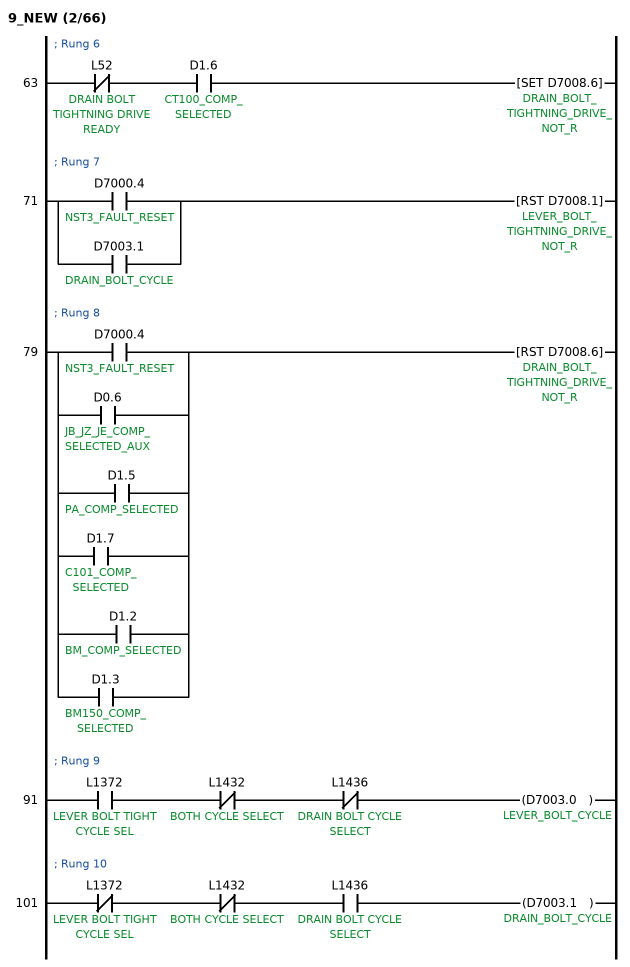
[picture p120: ladder of 9_NEW, rungs at steps 63 to 101]
; Rung 6
63    LDI     L52  ; DRAIN BOLT TIGHTNING DRIVE READY
      AND     D1.6  ; CT100_COMP_SELECTED
      SET     D7008.6  ; DRAIN_BOLT_TIGHTNING_DRIVE_NOT_R
; Rung 7
71    LD      D7000.4  ; NST3_FAULT_RESET
      OR      D7003.1  ; DRAIN_BOLT_CYCLE
      RST     D7008.1  ; LEVER_BOLT_TIGHTNING_DRIVE_NOT_R
; Rung 8
79    LD      D7000.4  ; NST3_FAULT_RESET
      OR      D0.6  ; JB_JZ_JE_COMP_SELECTED_AUX
      OR      D1.5  ; PA_COMP_SELECTED
      OR      D1.7  ; C101_COMP_SELECTED
      OR      D1.2  ; BM_COMP_SELECTED
      OR      D1.3  ; BM150_COMP_SELECTED
      RST     D7008.6  ; DRAIN_BOLT_TIGHTNING_DRIVE_NOT_R
; Rung 9
91    LD      L1372  ; LEVER BOLT TIGHT CYCLE SEL
      ANI     L1432  ; BOTH CYCLE SELECT
      ANI     L1436  ; DRAIN BOLT CYCLE SELECT
      OUT     D7003.0  ; LEVER_BOLT_CYCLE
; Rung 10
101   LDI     L1372  ; LEVER BOLT TIGHT CYCLE SEL
      ANI     L1432  ; BOTH CYCLE SELECT
      AND     L1436  ; DRAIN BOLT CYCLE SELECT
      OUT     D7003.1  ; DRAIN_BOLT_CYCLE
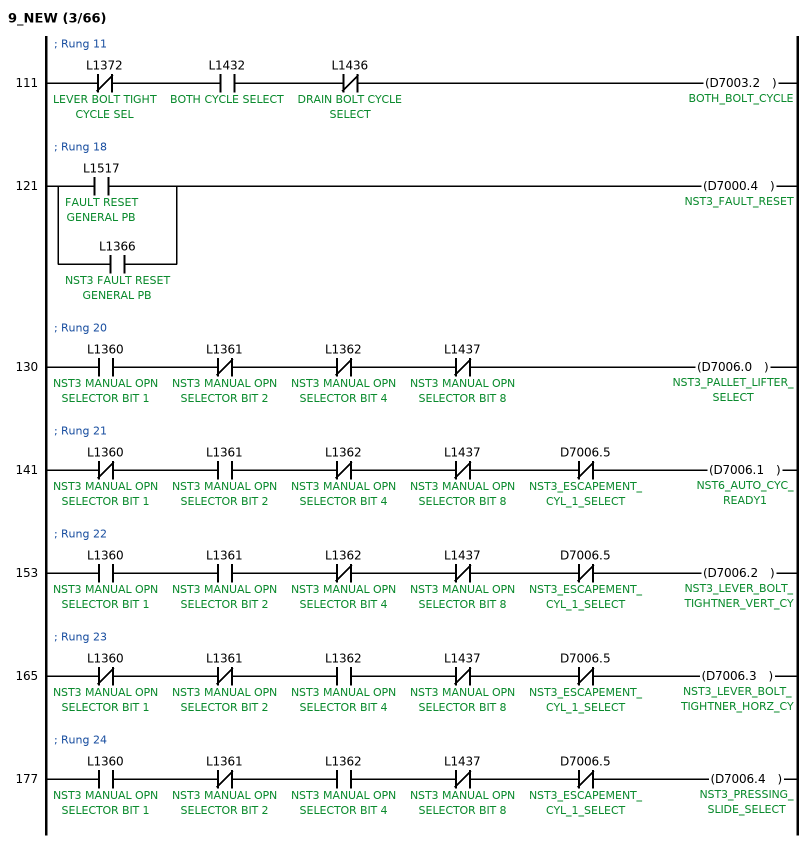
; Rung 11
111   LDI     L1372  ; LEVER BOLT TIGHT CYCLE SEL
      AND     L1432  ; BOTH CYCLE SELECT
      ANI     L1436  ; DRAIN BOLT CYCLE SELECT
      OUT     D7003.2  ; BOTH_BOLT_CYCLE
; Rung 18
121   LD      L1517  ; FAULT RESET GENERAL PB
      OR      L1366  ; NST3 FAULT RESET GENERAL PB
      OUT     D7000.4  ; NST3_FAULT_RESET
; Rung 20
130   LD      L1360  ; NST3 MANUAL OPN SELECTOR BIT 1
      ANI     L1361  ; NST3 MANUAL OPN SELECTOR BIT 2
      ANI     L1362  ; NST3 MANUAL OPN SELECTOR BIT 4
      ANI     L1437  ; NST3 MANUAL OPN SELECTOR BIT 8
      OUT     D7006.0  ; NST3_PALLET_LIFTER_SELECT
; Rung 21
141   LDI     L1360  ; NST3 MANUAL OPN SELECTOR BIT 1
      AND     L1361  ; NST3 MANUAL OPN SELECTOR BIT 2
      ANI     L1362  ; NST3 MANUAL OPN SELECTOR BIT 4
      ANI     L1437  ; NST3 MANUAL OPN SELECTOR BIT 8
      ANI     D7006.5  ; NST3_ESCAPEMENT_CYL_1_SELECT
      OUT     D7006.1  ; NST6_AUTO_CYC_READY1
; Rung 22
153   LD      L1360  ; NST3 MANUAL OPN SELECTOR BIT 1
      AND     L1361  ; NST3 MANUAL OPN SELECTOR BIT 2
      ANI     L1362  ; NST3 MANUAL OPN SELECTOR BIT 4
      ANI     L1437  ; NST3 MANUAL OPN SELECTOR BIT 8
      ANI     D7006.5  ; NST3_ESCAPEMENT_CYL_1_SELECT
      OUT     D7006.2  ; NST3_LEVER_BOLT_TIGHTNER_VERT_CY
; Rung 23
165   LDI     L1360  ; NST3 MANUAL OPN SELECTOR BIT 1
      ANI     L1361  ; NST3 MANUAL OPN SELECTOR BIT 2
      AND     L1362  ; NST3 MANUAL OPN SELECTOR BIT 4
      ANI     L1437  ; NST3 MANUAL OPN SELECTOR BIT 8
      ANI     D7006.5  ; NST3_ESCAPEMENT_CYL_1_SELECT
      OUT     D7006.3  ; NST3_LEVER_BOLT_TIGHTNER_HORZ_CY
; Rung 24
177   LD      L1360  ; NST3 MANUAL OPN SELECTOR BIT 1
      ANI     L1361  ; NST3 MANUAL OPN SELECTOR BIT 2
      AND     L1362  ; NST3 MANUAL OPN SELECTOR BIT 4
      ANI     L1437  ; NST3 MANUAL OPN SELECTOR BIT 8
      ANI     D7006.5  ; NST3_ESCAPEMENT_CYL_1_SELECT
      OUT     D7006.4  ; NST3_PRESSING_SLIDE_SELECT
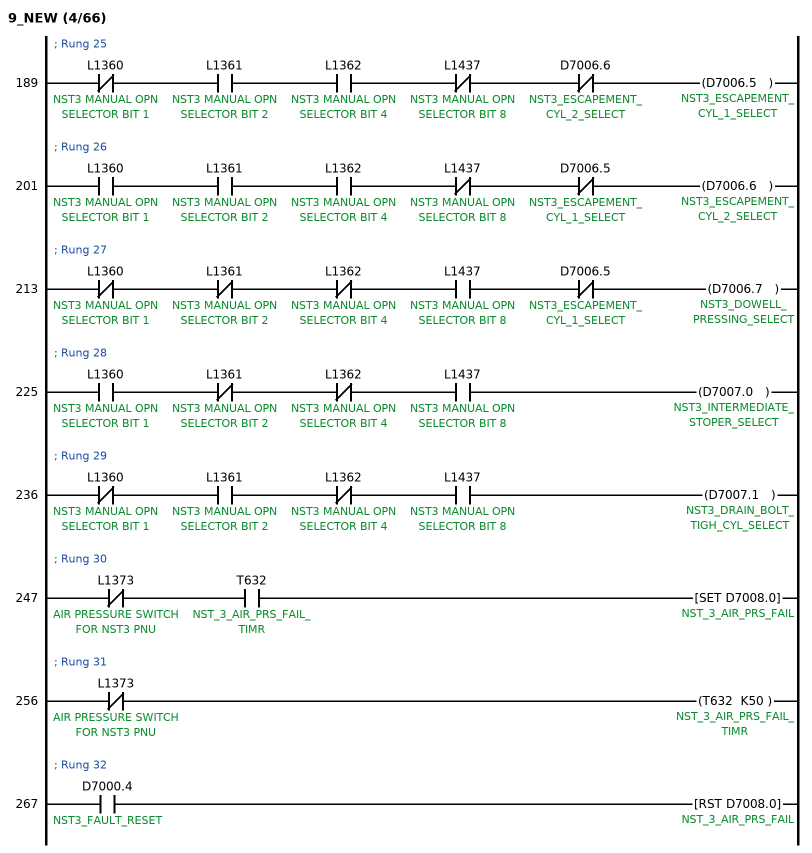
; Rung 25
189   LDI     L1360  ; NST3 MANUAL OPN SELECTOR BIT 1
      AND     L1361  ; NST3 MANUAL OPN SELECTOR BIT 2
      AND     L1362  ; NST3 MANUAL OPN SELECTOR BIT 4
      ANI     L1437  ; NST3 MANUAL OPN SELECTOR BIT 8
      ANI     D7006.6  ; NST3_ESCAPEMENT_CYL_2_SELECT
      OUT     D7006.5  ; NST3_ESCAPEMENT_CYL_1_SELECT
; Rung 26
201   LD      L1360  ; NST3 MANUAL OPN SELECTOR BIT 1
      AND     L1361  ; NST3 MANUAL OPN SELECTOR BIT 2
      AND     L1362  ; NST3 MANUAL OPN SELECTOR BIT 4
      ANI     L1437  ; NST3 MANUAL OPN SELECTOR BIT 8
      ANI     D7006.5  ; NST3_ESCAPEMENT_CYL_1_SELECT
      OUT     D7006.6  ; NST3_ESCAPEMENT_CYL_2_SELECT
; Rung 27
213   LDI     L1360  ; NST3 MANUAL OPN SELECTOR BIT 1
      ANI     L1361  ; NST3 MANUAL OPN SELECTOR BIT 2
      ANI     L1362  ; NST3 MANUAL OPN SELECTOR BIT 4
      AND     L1437  ; NST3 MANUAL OPN SELECTOR BIT 8
      ANI     D7006.5  ; NST3_ESCAPEMENT_CYL_1_SELECT
      OUT     D7006.7  ; NST3_DOWELL_PRESSING_SELECT
; Rung 28
225   LD      L1360  ; NST3 MANUAL OPN SELECTOR BIT 1
      ANI     L1361  ; NST3 MANUAL OPN SELECTOR BIT 2
      ANI     L1362  ; NST3 MANUAL OPN SELECTOR BIT 4
      AND     L1437  ; NST3 MANUAL OPN SELECTOR BIT 8
      OUT     D7007.0  ; NST3_INTERMEDIATE_STOPER_SELECT
; Rung 29
236   LDI     L1360  ; NST3 MANUAL OPN SELECTOR BIT 1
      AND     L1361  ; NST3 MANUAL OPN SELECTOR BIT 2
      ANI     L1362  ; NST3 MANUAL OPN SELECTOR BIT 4
      AND     L1437  ; NST3 MANUAL OPN SELECTOR BIT 8
      OUT     D7007.1  ; NST3_DRAIN_BOLT_TIGH_CYL_SELECT
; Rung 30
247   LDI     L1373  ; AIR PRESSURE SWITCH FOR NST3 PNU
      AND     T632  ; NST_3_AIR_PRS_FAIL_TIMR
      SET     D7008.0  ; NST_3_AIR_PRS_FAIL
; Rung 31
256   LDI     L1373  ; AIR PRESSURE SWITCH FOR NST3 PNU
      OUT     T632 K50  ; NST_3_AIR_PRS_FAIL_TIMR
; Rung 32
267   LD      D7000.4  ; NST3_FAULT_RESET
      RST     D7008.0  ; NST_3_AIR_PRS_FAIL
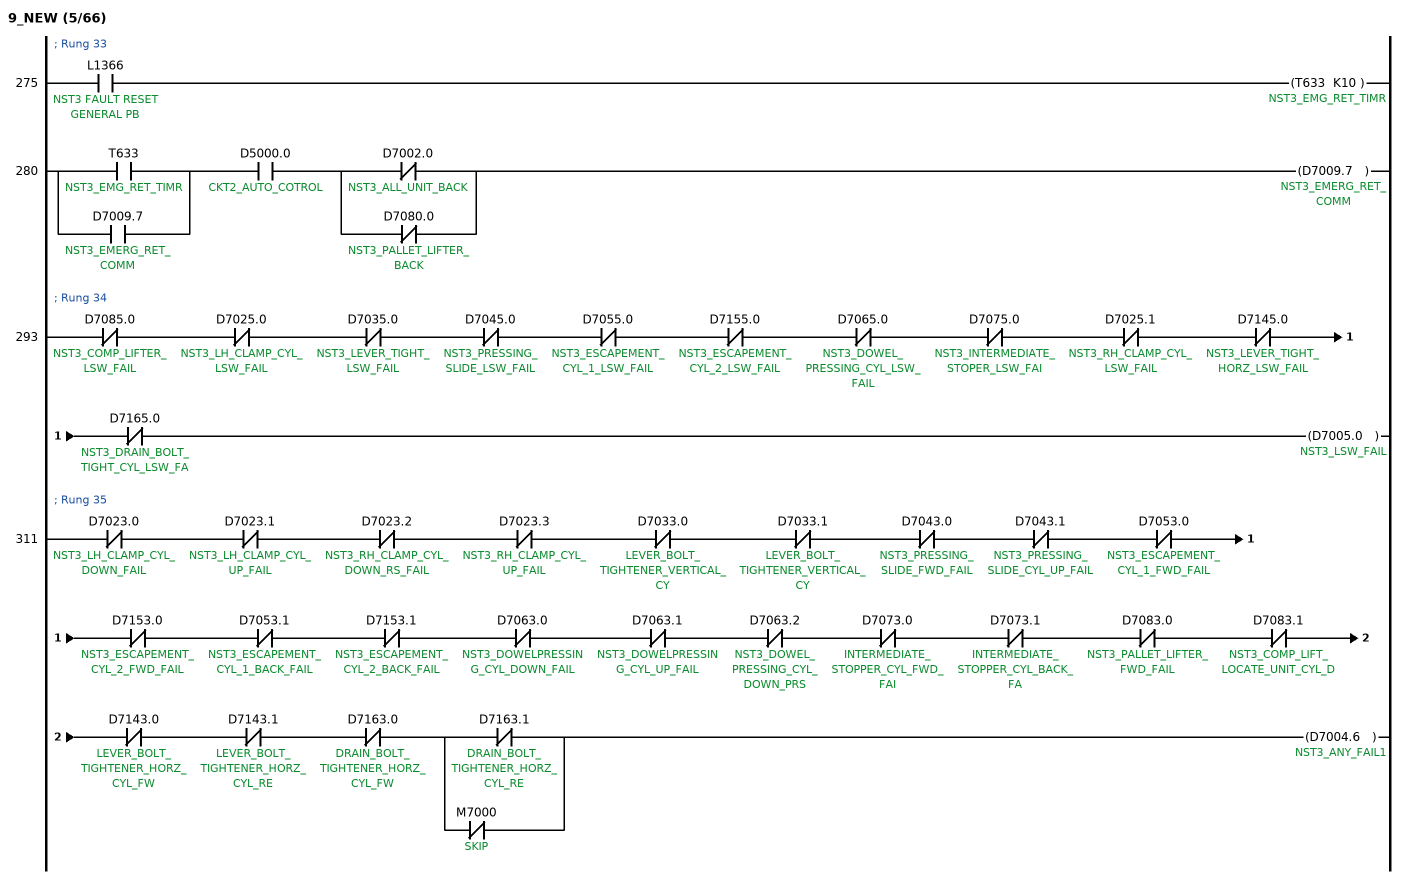
; Rung 33
275   LD      L1366  ; NST3 FAULT RESET GENERAL PB
      OUT     T633 K10  ; NST3_EMG_RET_TIMR
280   LD      T633  ; NST3_EMG_RET_TIMR
      OR      D7009.7  ; NST3_EMERG_RET_COMM
      AND     D5000.0  ; CKT2_AUTO_COTROL
      LDI     D7002.0  ; NST3_ALL_UNIT_BACK
      ORI     D7080.0  ; NST3_PALLET_LIFTER_BACK
      ANB
      OUT     D7009.7  ; NST3_EMERG_RET_COMM
; Rung 34
293   LDI     D7085.0  ; NST3_COMP_LIFTER_LSW_FAIL
      ANI     D7025.0  ; NST3_LH_CLAMP_CYL_LSW_FAIL
      ANI     D7035.0  ; NST3_LEVER_TIGHT_LSW_FAIL
      ANI     D7045.0  ; NST3_PRESSING_SLIDE_LSW_FAIL
      ANI     D7055.0  ; NST3_ESCAPEMENT_CYL_1_LSW_FAIL
      ANI     D7155.0  ; NST3_ESCAPEMENT_CYL_2_LSW_FAIL
      ANI     D7065.0  ; NST3_DOWEL_PRESSING_CYL_LSW_FAIL
      ANI     D7075.0  ; NST3_INTERMEDIATE_STOPER_LSW_FAI
      ANI     D7025.1  ; NST3_RH_CLAMP_CYL_LSW_FAIL
      ANI     D7145.0  ; NST3_LEVER_TIGHT_HORZ_LSW_FAIL
      ANI     D7165.0  ; NST3_DRAIN_BOLT_TIGHT_CYL_LSW_FA
      OUT     D7005.0  ; NST3_LSW_FAIL
; Rung 35
311   LDI     D7023.0  ; NST3_LH_CLAMP_CYL_DOWN_FAIL
      ANI     D7023.1  ; NST3_LH_CLAMP_CYL_UP_FAIL
      ANI     D7023.2  ; NST3_RH_CLAMP_CYL_DOWN_RS_FAIL
      ANI     D7023.3  ; NST3_RH_CLAMP_CYL_UP_FAIL
      ANI     D7033.0  ; LEVER_BOLT_TIGHTENER_VERTICAL_CY
      ANI     D7033.1  ; LEVER_BOLT_TIGHTENER_VERTICAL_CY
      ANI     D7043.0  ; NST3_PRESSING_SLIDE_FWD_FAIL
      ANI     D7043.1  ; NST3_PRESSING_SLIDE_CYL_UP_FAIL
      ANI     D7053.0  ; NST3_ESCAPEMENT_CYL_1_FWD_FAIL
      ANI     D7153.0  ; NST3_ESCAPEMENT_CYL_2_FWD_FAIL
      ANI     D7053.1  ; NST3_ESCAPEMENT_CYL_1_BACK_FAIL
      ANI     D7153.1  ; NST3_ESCAPEMENT_CYL_2_BACK_FAIL
      ANI     D7063.0  ; NST3_DOWELPRESSING_CYL_DOWN_FAIL
      ANI     D7063.1  ; NST3_DOWELPRESSING_CYL_UP_FAIL
      ANI     D7063.2  ; NST3_DOWEL_PRESSING_CYL_DOWN_PRS
      ANI     D7073.0  ; INTERMEDIATE_STOPPER_CYL_FWD_FAI
      ANI     D7073.1  ; INTERMEDIATE_STOPPER_CYL_BACK_FA
      ANI     D7083.0  ; NST3_PALLET_LIFTER_FWD_FAIL
      ANI     D7083.1  ; NST3_COMP_LIFT_LOCATE_UNIT_CYL_D
      ANI     D7143.0  ; LEVER_BOLT_TIGHTENER_HORZ_CYL_FW
      ANI     D7143.1  ; LEVER_BOLT_TIGHTENER_HORZ_CYL_RE
      ANI     D7163.0  ; DRAIN_BOLT_TIGHTENER_HORZ_CYL_FW
      LDI     D7163.1  ; DRAIN_BOLT_TIGHTENER_HORZ_CYL_RE
      ORI     M7000  ; SKIP
      ANB
      OUT     D7004.6  ; NST3_ANY_FAIL1
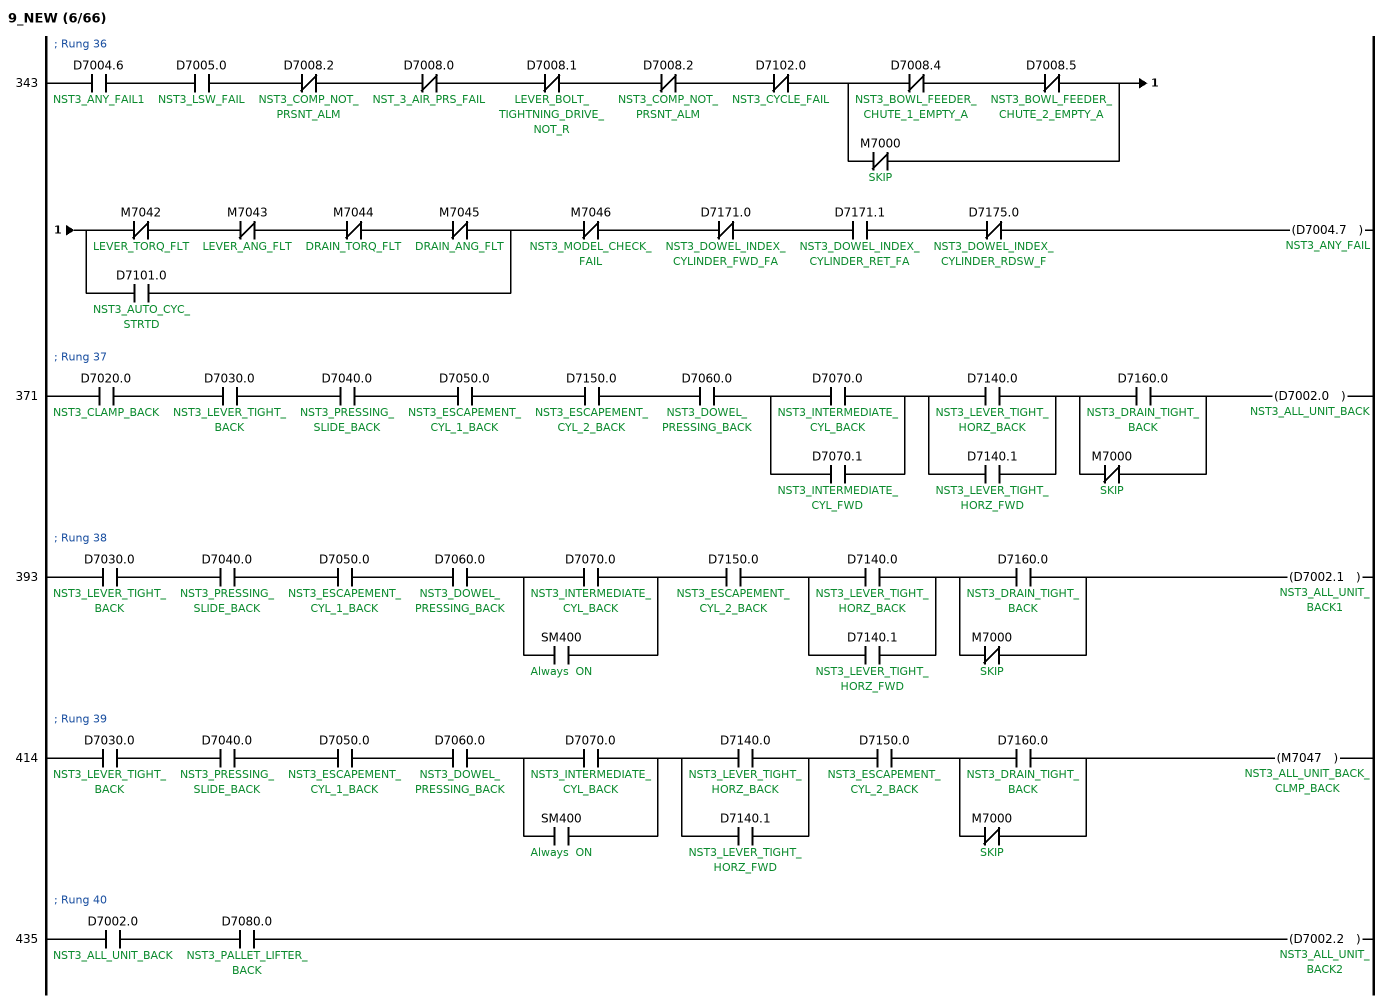
; Rung 36
343   LD      D7004.6  ; NST3_ANY_FAIL1
      AND     D7005.0  ; NST3_LSW_FAIL
      ANI     D7008.2  ; NST3_COMP_NOT_PRSNT_ALM
      ANI     D7008.0  ; NST_3_AIR_PRS_FAIL
      ANI     D7008.1  ; LEVER_BOLT_TIGHTNING_DRIVE_NOT_R
      ANI     D7008.2  ; NST3_COMP_NOT_PRSNT_ALM
      ANI     D7102.0  ; NST3_CYCLE_FAIL
      LDI     D7008.4  ; NST3_BOWL_FEEDER_CHUTE_1_EMPTY_A
      ANI     D7008.5  ; NST3_BOWL_FEEDER_CHUTE_2_EMPTY_A
      ORI     M7000  ; SKIP
      ANB
      LDI     M7042  ; LEVER_TORQ_FLT
      ANI     M7043  ; LEVER_ANG_FLT
      ANI     M7044  ; DRAIN_TORQ_FLT
      ANI     M7045  ; DRAIN_ANG_FLT
      OR      D7101.0  ; NST3_AUTO_CYC_STRTD
      ANB
      ANI     M7046  ; NST3_MODEL_CHECK_FAIL
      ANI     D7171.0  ; NST3_DOWEL_INDEX_CYLINDER_FWD_FA
      AND     D7171.1  ; NST3_DOWEL_INDEX_CYLINDER_RET_FA
      ANI     D7175.0  ; NST3_DOWEL_INDEX_CYLINDER_RDSW_F
      OUT     D7004.7  ; NST3_ANY_FAIL
; Rung 37
371   LD      D7020.0  ; NST3_CLAMP_BACK
      AND     D7030.0  ; NST3_LEVER_TIGHT_BACK
      AND     D7040.0  ; NST3_PRESSING_SLIDE_BACK
      AND     D7050.0  ; NST3_ESCAPEMENT_CYL_1_BACK
      AND     D7150.0  ; NST3_ESCAPEMENT_CYL_2_BACK
      AND     D7060.0  ; NST3_DOWEL_PRESSING_BACK
      LD      D7070.0  ; NST3_INTERMEDIATE_CYL_BACK
      OR      D7070.1  ; NST3_INTERMEDIATE_CYL_FWD
      ANB
      LD      D7140.0  ; NST3_LEVER_TIGHT_HORZ_BACK
      OR      D7140.1  ; NST3_LEVER_TIGHT_HORZ_FWD
      ANB
      LD      D7160.0  ; NST3_DRAIN_TIGHT_BACK
      ORI     M7000  ; SKIP
      ANB
      OUT     D7002.0  ; NST3_ALL_UNIT_BACK
; Rung 38
393   LD      D7030.0  ; NST3_LEVER_TIGHT_BACK
      AND     D7040.0  ; NST3_PRESSING_SLIDE_BACK
      AND     D7050.0  ; NST3_ESCAPEMENT_CYL_1_BACK
      AND     D7060.0  ; NST3_DOWEL_PRESSING_BACK
      LD      D7070.0  ; NST3_INTERMEDIATE_CYL_BACK
      OR      SM400  ; Always  ON
      ANB
      AND     D7150.0  ; NST3_ESCAPEMENT_CYL_2_BACK
      LD      D7140.0  ; NST3_LEVER_TIGHT_HORZ_BACK
      OR      D7140.1  ; NST3_LEVER_TIGHT_HORZ_FWD
      ANB
      LD      D7160.0  ; NST3_DRAIN_TIGHT_BACK
      ORI     M7000  ; SKIP
      ANB
      OUT     D7002.1  ; NST3_ALL_UNIT_BACK1
; Rung 39
414   LD      D7030.0  ; NST3_LEVER_TIGHT_BACK
      AND     D7040.0  ; NST3_PRESSING_SLIDE_BACK
      AND     D7050.0  ; NST3_ESCAPEMENT_CYL_1_BACK
      AND     D7060.0  ; NST3_DOWEL_PRESSING_BACK
      LD      D7070.0  ; NST3_INTERMEDIATE_CYL_BACK
      OR      SM400  ; Always  ON
      ANB
      LD      D7140.0  ; NST3_LEVER_TIGHT_HORZ_BACK
      OR      D7140.1  ; NST3_LEVER_TIGHT_HORZ_FWD
      ANB
      AND     D7150.0  ; NST3_ESCAPEMENT_CYL_2_BACK
      LD      D7160.0  ; NST3_DRAIN_TIGHT_BACK
      ORI     M7000  ; SKIP
      ANB
      OUT     M7047  ; NST3_ALL_UNIT_BACK_CLMP_BACK
; Rung 40
435   LD      D7002.0  ; NST3_ALL_UNIT_BACK
      AND     D7080.0  ; NST3_PALLET_LIFTER_BACK
      OUT     D7002.2  ; NST3_ALL_UNIT_BACK2
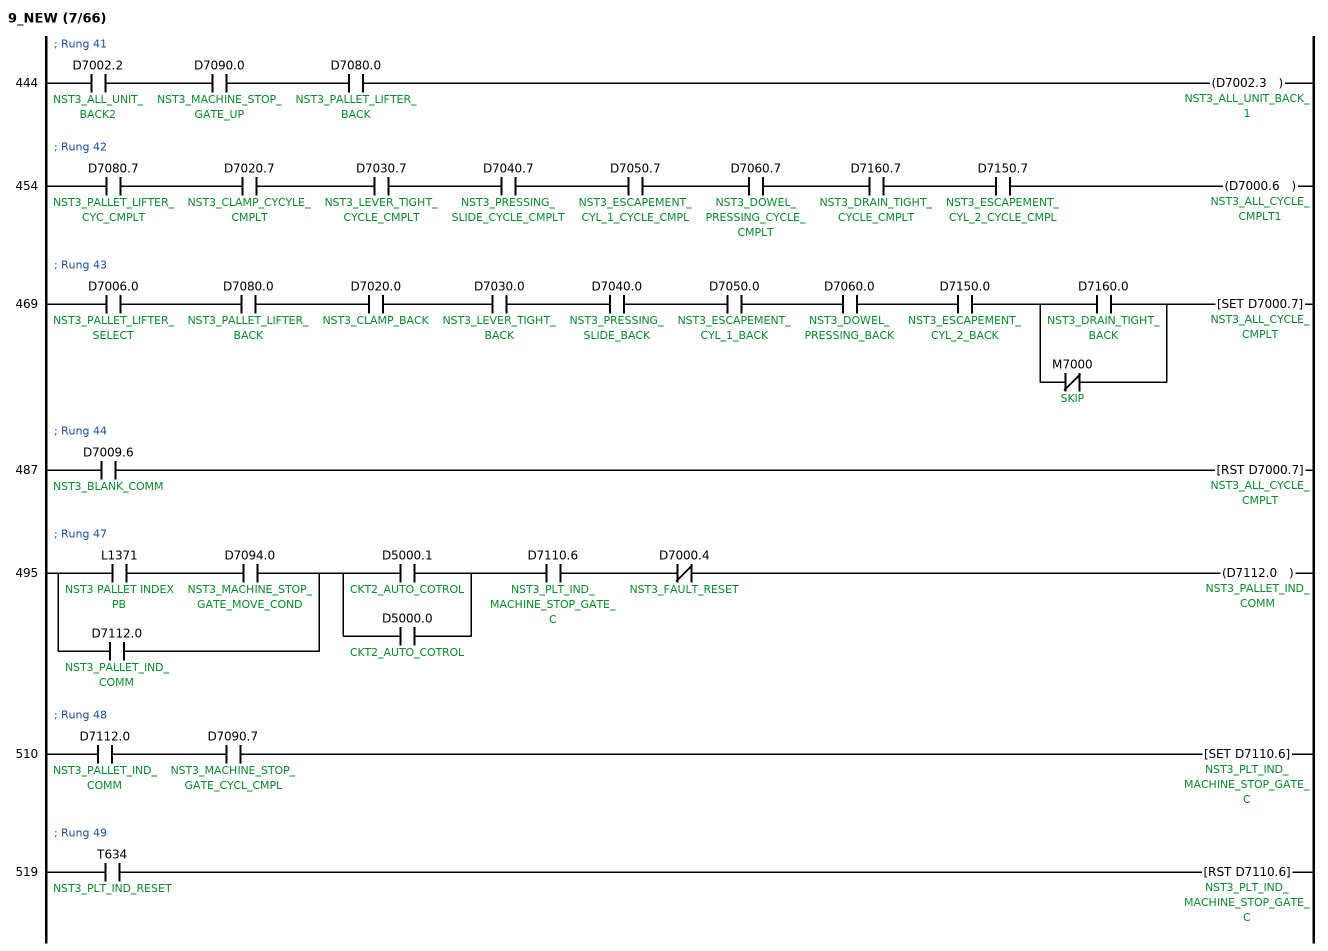
; Rung 41
444   LD      D7002.2  ; NST3_ALL_UNIT_BACK2
      AND     D7090.0  ; NST3_MACHINE_STOP_GATE_UP
      AND     D7080.0  ; NST3_PALLET_LIFTER_BACK
      OUT     D7002.3  ; NST3_ALL_UNIT_BACK_1
; Rung 42
454   LD      D7080.7  ; NST3_PALLET_LIFTER_CYC_CMPLT
      AND     D7020.7  ; NST3_CLAMP_CYCYLE_CMPLT
      AND     D7030.7  ; NST3_LEVER_TIGHT_CYCLE_CMPLT
      AND     D7040.7  ; NST3_PRESSING_SLIDE_CYCLE_CMPLT
      AND     D7050.7  ; NST3_ESCAPEMENT_CYL_1_CYCLE_CMPL
      AND     D7060.7  ; NST3_DOWEL_PRESSING_CYCLE_CMPLT
      AND     D7160.7  ; NST3_DRAIN_TIGHT_CYCLE_CMPLT
      AND     D7150.7  ; NST3_ESCAPEMENT_CYL_2_CYCLE_CMPL
      OUT     D7000.6  ; NST3_ALL_CYCLE_CMPLT1
; Rung 43
469   LD      D7006.0  ; NST3_PALLET_LIFTER_SELECT
      AND     D7080.0  ; NST3_PALLET_LIFTER_BACK
      AND     D7020.0  ; NST3_CLAMP_BACK
      AND     D7030.0  ; NST3_LEVER_TIGHT_BACK
      AND     D7040.0  ; NST3_PRESSING_SLIDE_BACK
      AND     D7050.0  ; NST3_ESCAPEMENT_CYL_1_BACK
      AND     D7060.0  ; NST3_DOWEL_PRESSING_BACK
      AND     D7150.0  ; NST3_ESCAPEMENT_CYL_2_BACK
      LD      D7160.0  ; NST3_DRAIN_TIGHT_BACK
      ORI     M7000  ; SKIP
      ANB
      SET     D7000.7  ; NST3_ALL_CYCLE_CMPLT
; Rung 44
487   LD      D7009.6  ; NST3_BLANK_COMM
      RST     D7000.7  ; NST3_ALL_CYCLE_CMPLT
; Rung 47
495   LD      L1371  ; NST3 PALLET INDEX PB
      AND     D7094.0  ; NST3_MACHINE_STOP_GATE_MOVE_COND
      OR      D7112.0  ; NST3_PALLET_IND_COMM
      LD      D5000.1  ; CKT2_AUTO_COTROL
      OR      D5000.0  ; CKT2_AUTO_COTROL
      ANB
      AND     D7110.6  ; NST3_PLT_IND_MACHINE_STOP_GATE_C
      ANI     D7000.4  ; NST3_FAULT_RESET
      OUT     D7112.0  ; NST3_PALLET_IND_COMM
; Rung 48
510   LD      D7112.0  ; NST3_PALLET_IND_COMM
      AND     D7090.7  ; NST3_MACHINE_STOP_GATE_CYCL_CMPL
      SET     D7110.6  ; NST3_PLT_IND_MACHINE_STOP_GATE_C
; Rung 49
519   LD      T634  ; NST3_PLT_IND_RESET
      RST     D7110.6  ; NST3_PLT_IND_MACHINE_STOP_GATE_C
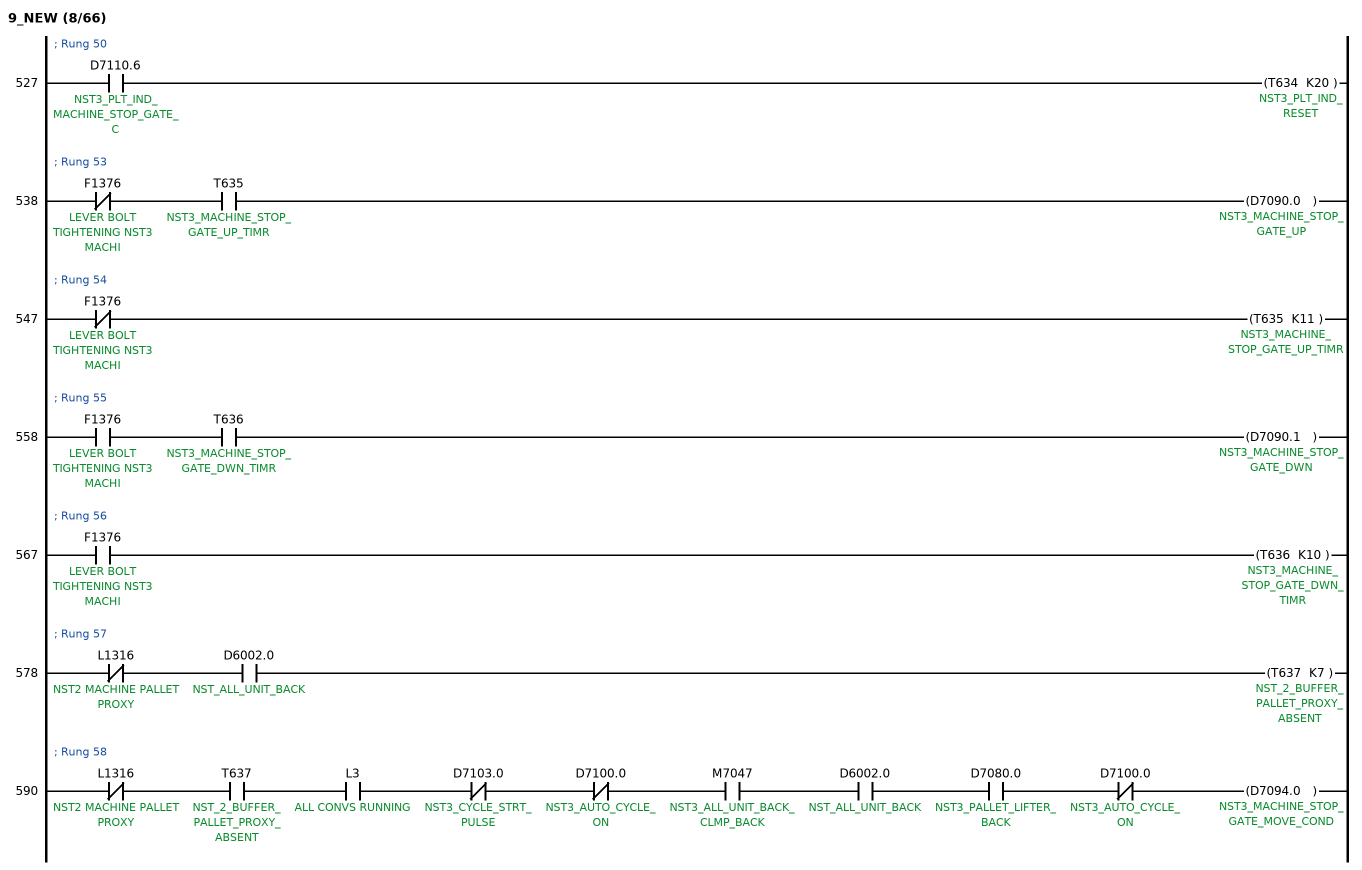
; Rung 50
527   LD      D7110.6  ; NST3_PLT_IND_MACHINE_STOP_GATE_C
      OUT     T634 K20  ; NST3_PLT_IND_RESET
; Rung 53
538   LDI     F1376  ; LEVER BOLT TIGHTENING NST3 MACHI
      AND     T635  ; NST3_MACHINE_STOP_GATE_UP_TIMR
      OUT     D7090.0  ; NST3_MACHINE_STOP_GATE_UP
; Rung 54
547   LDI     F1376  ; LEVER BOLT TIGHTENING NST3 MACHI
      OUT     T635 K11  ; NST3_MACHINE_STOP_GATE_UP_TIMR
; Rung 55
558   LD      F1376  ; LEVER BOLT TIGHTENING NST3 MACHI
      AND     T636  ; NST3_MACHINE_STOP_GATE_DWN_TIMR
      OUT     D7090.1  ; NST3_MACHINE_STOP_GATE_DWN
; Rung 56
567   LD      F1376  ; LEVER BOLT TIGHTENING NST3 MACHI
      OUT     T636 K10  ; NST3_MACHINE_STOP_GATE_DWN_TIMR
; Rung 57
578   LDI     L1316  ; NST2 MACHINE PALLET PROXY
      AND     D6002.0  ; NST_ALL_UNIT_BACK
      OUT     T637 K7  ; NST_2_BUFFER_PALLET_PROXY_ABSENT
; Rung 58
590   LDI     L1316  ; NST2 MACHINE PALLET PROXY
      AND     T637  ; NST_2_BUFFER_PALLET_PROXY_ABSENT
      AND     L3  ; ALL CONVS RUNNING
      ANI     D7103.0  ; NST3_CYCLE_STRT_PULSE
      ANI     D7100.0  ; NST3_AUTO_CYCLE_ON
      AND     M7047  ; NST3_ALL_UNIT_BACK_CLMP_BACK
      AND     D6002.0  ; NST_ALL_UNIT_BACK
      AND     D7080.0  ; NST3_PALLET_LIFTER_BACK
      ANI     D7100.0  ; NST3_AUTO_CYCLE_ON
      OUT     D7094.0  ; NST3_MACHINE_STOP_GATE_MOVE_COND
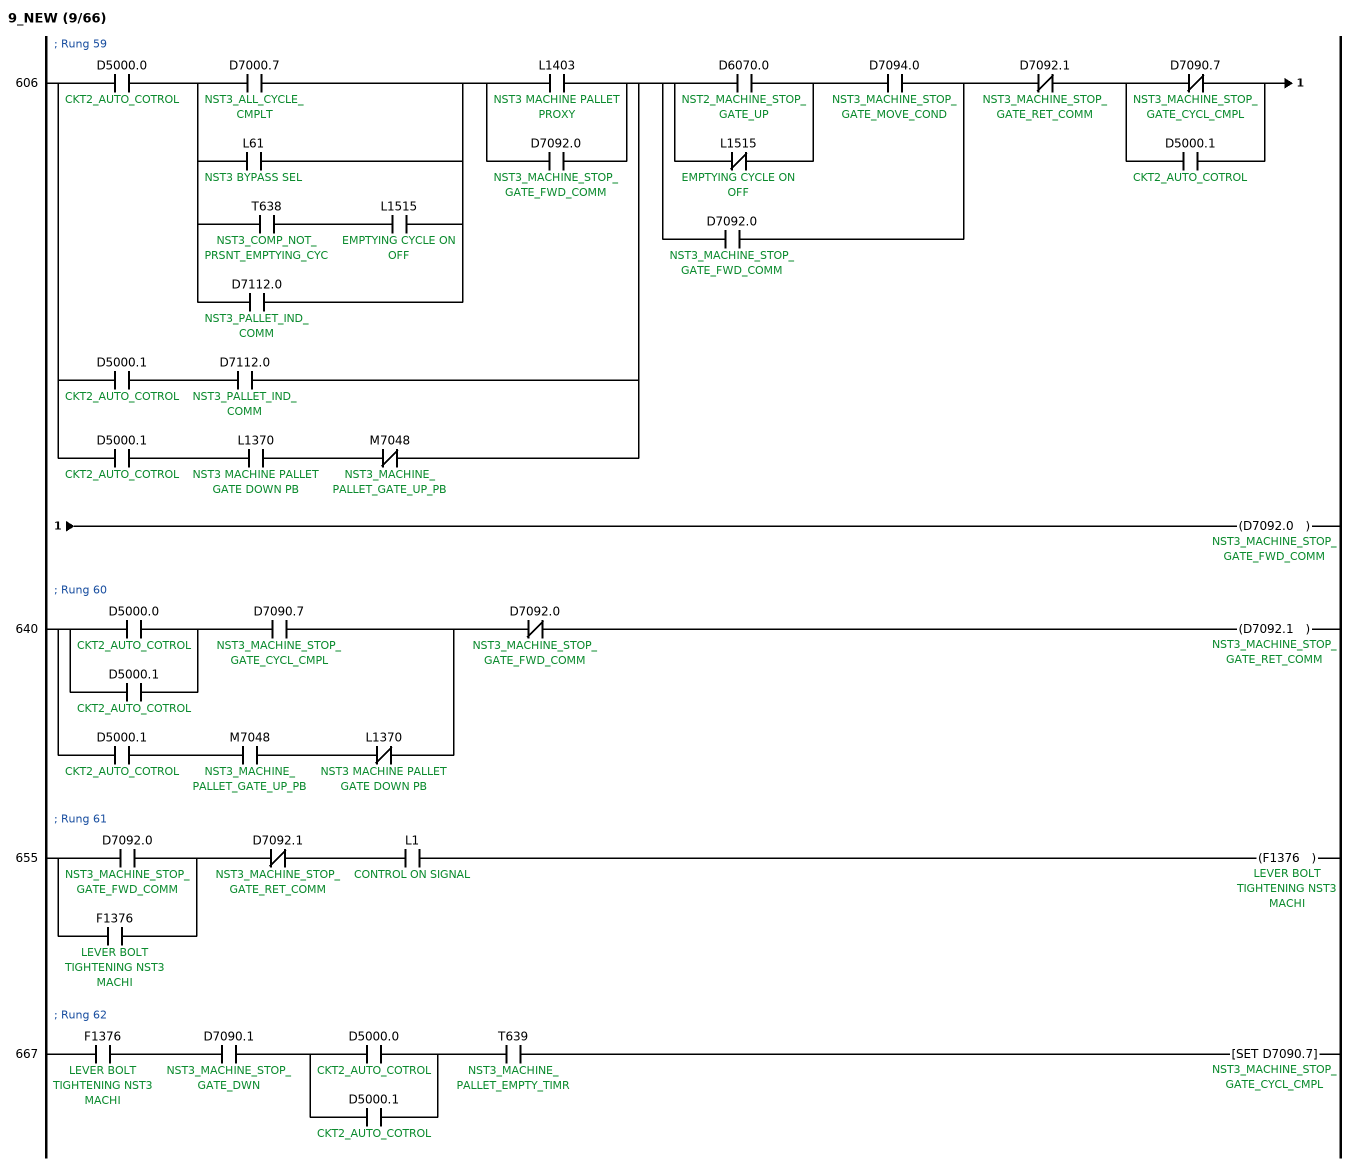
; Rung 59
606   LD      D5000.0  ; CKT2_AUTO_COTROL
      LD      D7000.7  ; NST3_ALL_CYCLE_CMPLT
      OR      L61  ; NST3 BYPASS SEL
      LD      T638  ; NST3_COMP_NOT_PRSNT_EMPTYING_CYC
      AND     L1515  ; EMPTYING CYCLE ON OFF
      ORB
      OR      D7112.0  ; NST3_PALLET_IND_COMM
      ANB
      LD      L1403  ; NST3 MACHINE PALLET PROXY
      OR      D7092.0  ; NST3_MACHINE_STOP_GATE_FWD_COMM
      ANB
      LD      D5000.1  ; CKT2_AUTO_COTROL
      AND     D7112.0  ; NST3_PALLET_IND_COMM
      ORB
      LD      D5000.1  ; CKT2_AUTO_COTROL
      AND     L1370  ; NST3 MACHINE PALLET GATE DOWN PB
      ANI     M7048  ; NST3_MACHINE_PALLET_GATE_UP_PB
      ORB
      LD      D6070.0  ; NST2_MACHINE_STOP_GATE_UP
      ORI     L1515  ; EMPTYING CYCLE ON OFF
      AND     D7094.0  ; NST3_MACHINE_STOP_GATE_MOVE_COND
      OR      D7092.0  ; NST3_MACHINE_STOP_GATE_FWD_COMM
      ANB
      ANI     D7092.1  ; NST3_MACHINE_STOP_GATE_RET_COMM
      LDI     D7090.7  ; NST3_MACHINE_STOP_GATE_CYCL_CMPL
      OR      D5000.1  ; CKT2_AUTO_COTROL
      ANB
      OUT     D7092.0  ; NST3_MACHINE_STOP_GATE_FWD_COMM
; Rung 60
640   LD      D5000.0  ; CKT2_AUTO_COTROL
      OR      D5000.1  ; CKT2_AUTO_COTROL
      AND     D7090.7  ; NST3_MACHINE_STOP_GATE_CYCL_CMPL
      LD      D5000.1  ; CKT2_AUTO_COTROL
      AND     M7048  ; NST3_MACHINE_PALLET_GATE_UP_PB
      ANI     L1370  ; NST3 MACHINE PALLET GATE DOWN PB
      ORB
      ANI     D7092.0  ; NST3_MACHINE_STOP_GATE_FWD_COMM
      OUT     D7092.1  ; NST3_MACHINE_STOP_GATE_RET_COMM
; Rung 61
655   LD      D7092.0  ; NST3_MACHINE_STOP_GATE_FWD_COMM
      OR      F1376  ; LEVER BOLT TIGHTENING NST3 MACHI
      ANI     D7092.1  ; NST3_MACHINE_STOP_GATE_RET_COMM
      AND     L1  ; CONTROL ON SIGNAL
      OUT     F1376  ; LEVER BOLT TIGHTENING NST3 MACHI
; Rung 62
667   LD      F1376  ; LEVER BOLT TIGHTENING NST3 MACHI
      AND     D7090.1  ; NST3_MACHINE_STOP_GATE_DWN
      LD      D5000.0  ; CKT2_AUTO_COTROL
      OR      D5000.1  ; CKT2_AUTO_COTROL
      ANB
      AND     T639  ; NST3_MACHINE_PALLET_EMPTY_TIMR
      SET     D7090.7  ; NST3_MACHINE_STOP_GATE_CYCL_CMPL
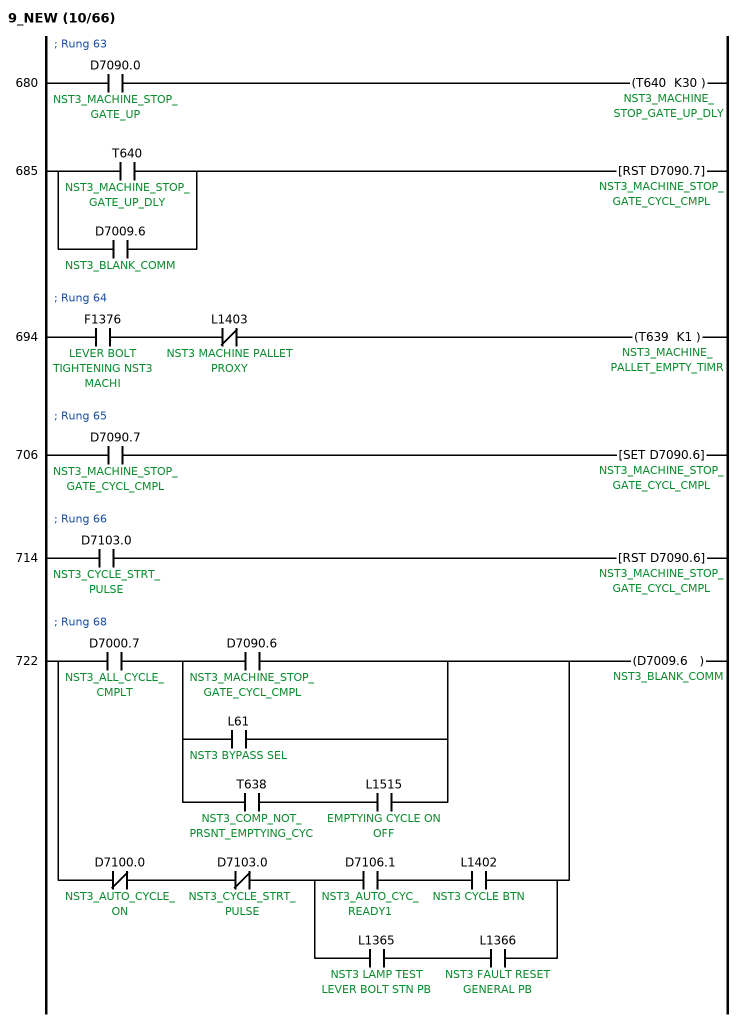
; Rung 63
680   LD      D7090.0  ; NST3_MACHINE_STOP_GATE_UP
      OUT     T640 K30  ; NST3_MACHINE_STOP_GATE_UP_DLY
685   LD      T640  ; NST3_MACHINE_STOP_GATE_UP_DLY
      OR      D7009.6  ; NST3_BLANK_COMM
      RST     D7090.7  ; NST3_MACHINE_STOP_GATE_CYCL_CMPL
; Rung 64
694   LD      F1376  ; LEVER BOLT TIGHTENING NST3 MACHI
      ANI     L1403  ; NST3 MACHINE PALLET PROXY
      OUT     T639 K1  ; NST3_MACHINE_PALLET_EMPTY_TIMR
; Rung 65
706   LD      D7090.7  ; NST3_MACHINE_STOP_GATE_CYCL_CMPL
      SET     D7090.6  ; NST3_MACHINE_STOP_GATE_CYCL_CMPL
; Rung 66
714   LD      D7103.0  ; NST3_CYCLE_STRT_PULSE
      RST     D7090.6  ; NST3_MACHINE_STOP_GATE_CYCL_CMPL
; Rung 68
722   LD      D7000.7  ; NST3_ALL_CYCLE_CMPLT
      LD      D7090.6  ; NST3_MACHINE_STOP_GATE_CYCL_CMPL
      OR      L61  ; NST3 BYPASS SEL
      LD      T638  ; NST3_COMP_NOT_PRSNT_EMPTYING_CYC
      AND     L1515  ; EMPTYING CYCLE ON OFF
      ORB
      ANB
      LDI     D7100.0  ; NST3_AUTO_CYCLE_ON
      ANI     D7103.0  ; NST3_CYCLE_STRT_PULSE
      LD      D7106.1  ; NST3_AUTO_CYC_READY1
      AND     L1402  ; NST3 CYCLE BTN
      LD      L1365  ; NST3 LAMP TEST LEVER BOLT STN PB
      AND     L1366  ; NST3 FAULT RESET GENERAL PB
      ORB
      ANB
      ORB
      OUT     D7009.6  ; NST3_BLANK_COMM
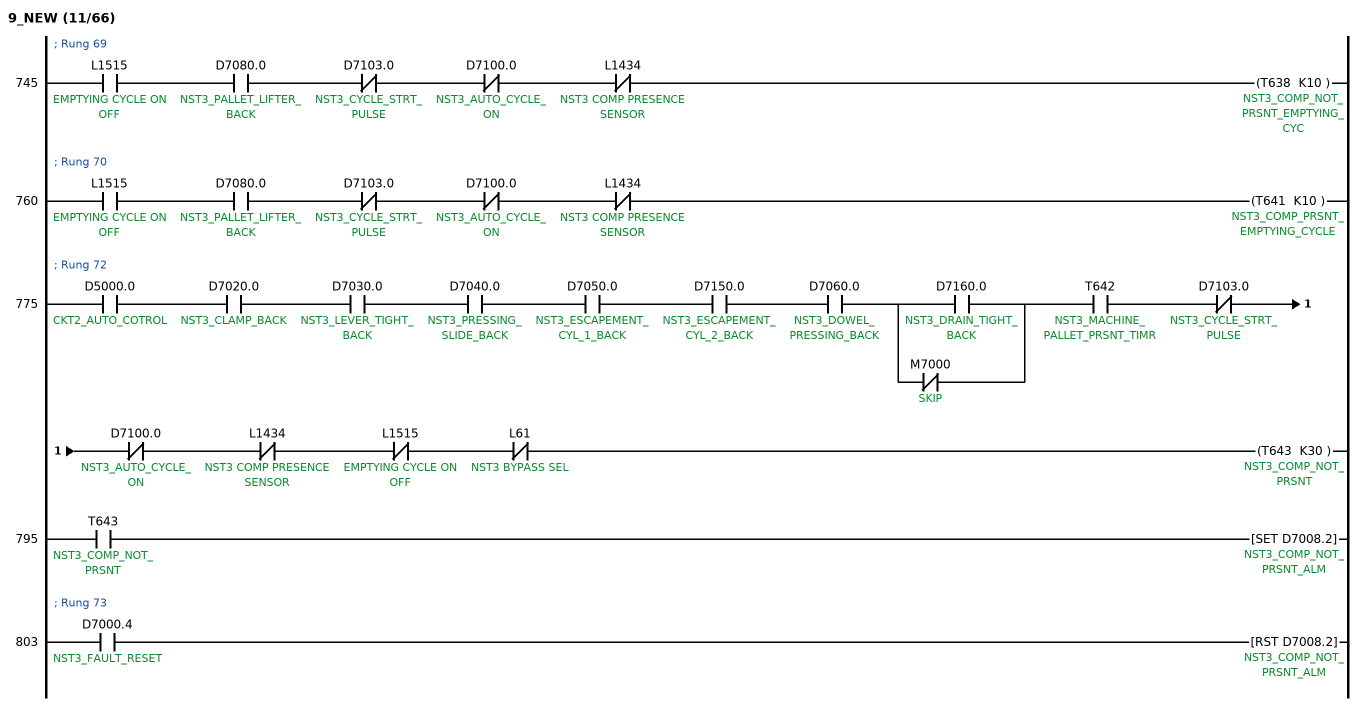
; Rung 69
745   LD      L1515  ; EMPTYING CYCLE ON OFF
      AND     D7080.0  ; NST3_PALLET_LIFTER_BACK
      ANI     D7103.0  ; NST3_CYCLE_STRT_PULSE
      ANI     D7100.0  ; NST3_AUTO_CYCLE_ON
      ANI     L1434  ; NST3 COMP PRESENCE SENSOR
      OUT     T638 K10  ; NST3_COMP_NOT_PRSNT_EMPTYING_CYC
; Rung 70
760   LD      L1515  ; EMPTYING CYCLE ON OFF
      AND     D7080.0  ; NST3_PALLET_LIFTER_BACK
      ANI     D7103.0  ; NST3_CYCLE_STRT_PULSE
      ANI     D7100.0  ; NST3_AUTO_CYCLE_ON
      ANI     L1434  ; NST3 COMP PRESENCE SENSOR
      OUT     T641 K10  ; NST3_COMP_PRSNT_EMPTYING_CYCLE
; Rung 72
775   LD      D5000.0  ; CKT2_AUTO_COTROL
      AND     D7020.0  ; NST3_CLAMP_BACK
      AND     D7030.0  ; NST3_LEVER_TIGHT_BACK
      AND     D7040.0  ; NST3_PRESSING_SLIDE_BACK
      AND     D7050.0  ; NST3_ESCAPEMENT_CYL_1_BACK
      AND     D7150.0  ; NST3_ESCAPEMENT_CYL_2_BACK
      AND     D7060.0  ; NST3_DOWEL_PRESSING_BACK
      LD      D7160.0  ; NST3_DRAIN_TIGHT_BACK
      ORI     M7000  ; SKIP
      ANB
      AND     T642  ; NST3_MACHINE_PALLET_PRSNT_TIMR
      ANI     D7103.0  ; NST3_CYCLE_STRT_PULSE
      ANI     D7100.0  ; NST3_AUTO_CYCLE_ON
      ANI     L1434  ; NST3 COMP PRESENCE SENSOR
      ANI     L1515  ; EMPTYING CYCLE ON OFF
      ANI     L61  ; NST3 BYPASS SEL
      OUT     T643 K30  ; NST3_COMP_NOT_PRSNT
795   LD      T643  ; NST3_COMP_NOT_PRSNT
      SET     D7008.2  ; NST3_COMP_NOT_PRSNT_ALM
; Rung 73
803   LD      D7000.4  ; NST3_FAULT_RESET
      RST     D7008.2  ; NST3_COMP_NOT_PRSNT_ALM
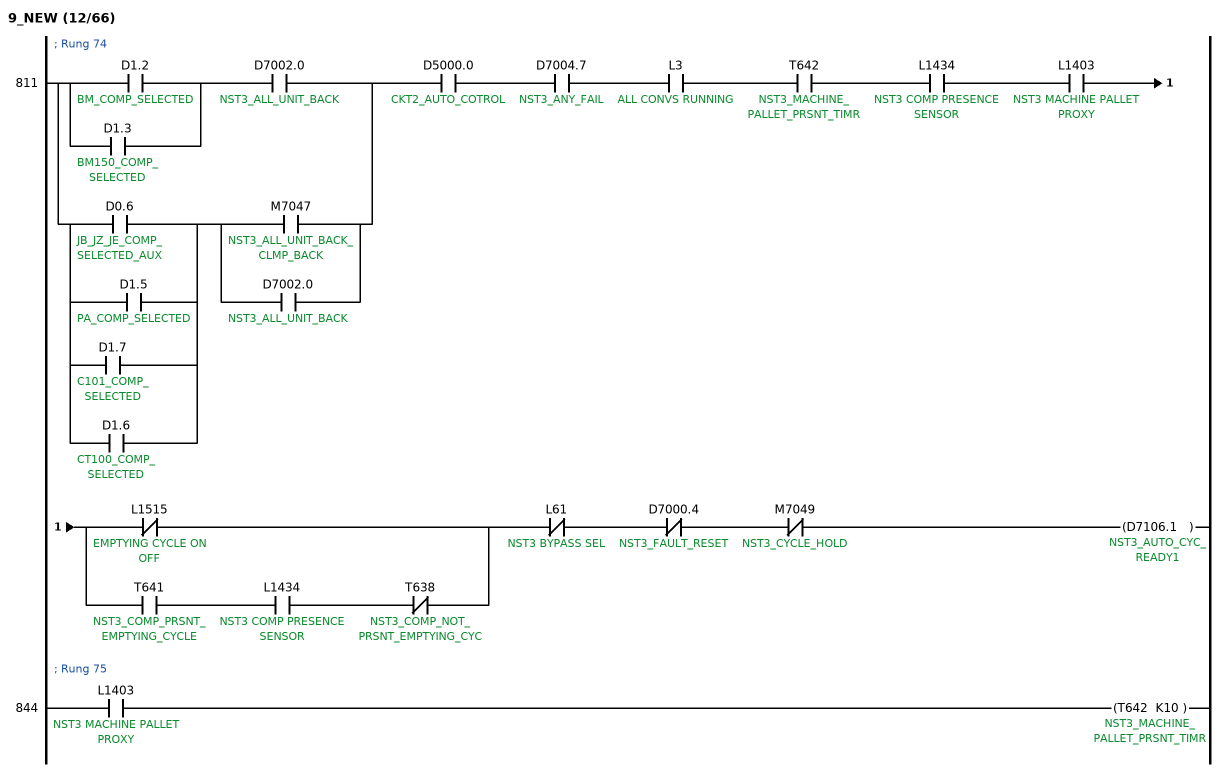
; Rung 74
811   LD      D1.2  ; BM_COMP_SELECTED
      OR      D1.3  ; BM150_COMP_SELECTED
      AND     D7002.0  ; NST3_ALL_UNIT_BACK
      LD      D0.6  ; JB_JZ_JE_COMP_SELECTED_AUX
      OR      D1.5  ; PA_COMP_SELECTED
      OR      D1.7  ; C101_COMP_SELECTED
      OR      D1.6  ; CT100_COMP_SELECTED
      LD      M7047  ; NST3_ALL_UNIT_BACK_CLMP_BACK
      OR      D7002.0  ; NST3_ALL_UNIT_BACK
      ANB
      ORB
      AND     D5000.0  ; CKT2_AUTO_COTROL
      AND     D7004.7  ; NST3_ANY_FAIL
      AND     L3  ; ALL CONVS RUNNING
      AND     T642  ; NST3_MACHINE_PALLET_PRSNT_TIMR
      AND     L1434  ; NST3 COMP PRESENCE SENSOR
      AND     L1403  ; NST3 MACHINE PALLET PROXY
      LDI     L1515  ; EMPTYING CYCLE ON OFF
      LD      T641  ; NST3_COMP_PRSNT_EMPTYING_CYCLE
      AND     L1434  ; NST3 COMP PRESENCE SENSOR
      ANI     T638  ; NST3_COMP_NOT_PRSNT_EMPTYING_CYC
      ORB
      ANB
      ANI     L61  ; NST3 BYPASS SEL
      ANI     D7000.4  ; NST3_FAULT_RESET
      ANI     M7049  ; NST3_CYCLE_HOLD
      OUT     D7106.1  ; NST3_AUTO_CYC_READY1
; Rung 75
844   LD      L1403  ; NST3 MACHINE PALLET PROXY
      OUT     T642 K10  ; NST3_MACHINE_PALLET_PRSNT_TIMR
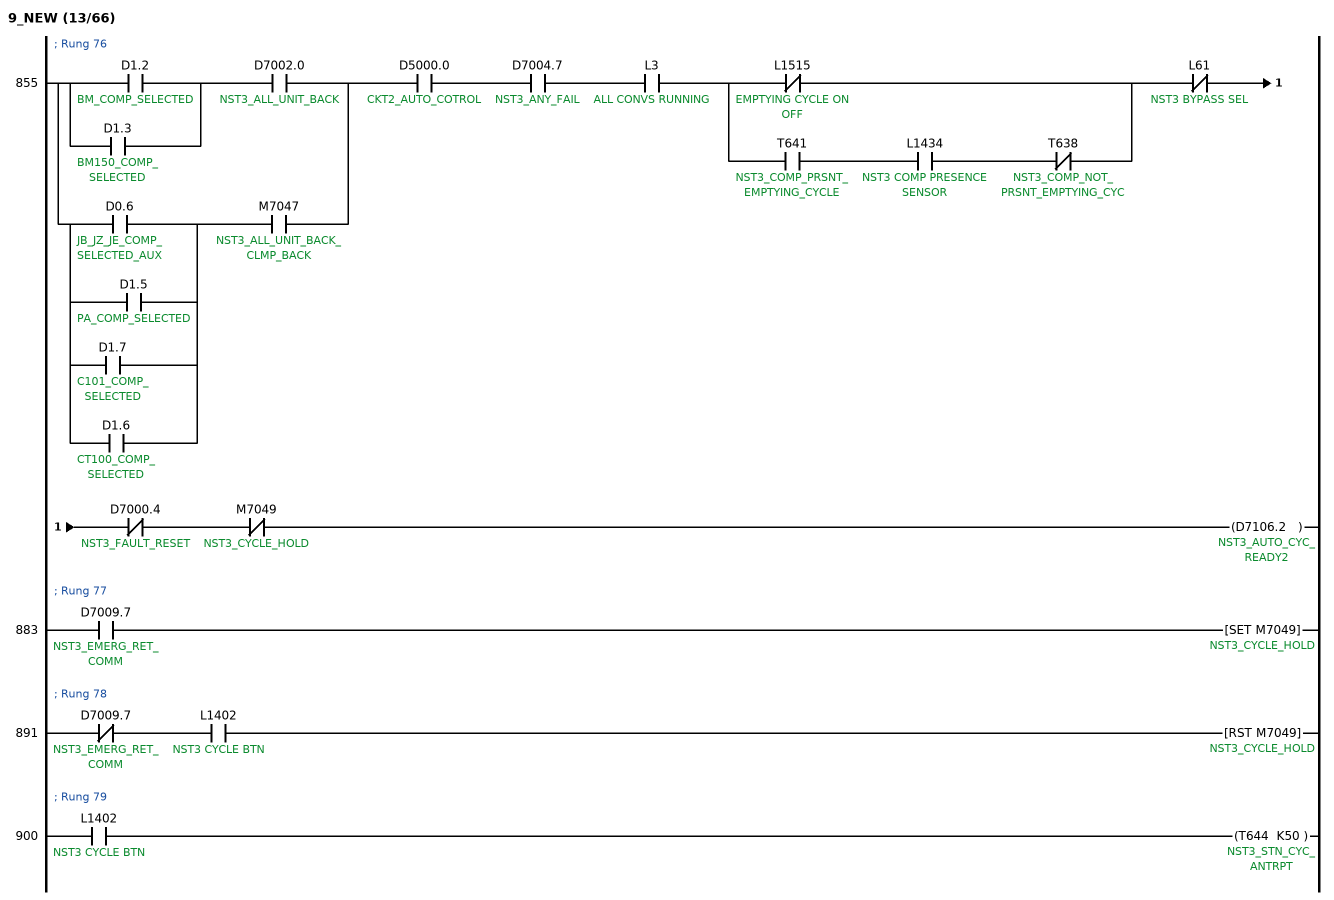
; Rung 76
855   LD      D1.2  ; BM_COMP_SELECTED
      OR      D1.3  ; BM150_COMP_SELECTED
      AND     D7002.0  ; NST3_ALL_UNIT_BACK
      LD      D0.6  ; JB_JZ_JE_COMP_SELECTED_AUX
      OR      D1.5  ; PA_COMP_SELECTED
      OR      D1.7  ; C101_COMP_SELECTED
      OR      D1.6  ; CT100_COMP_SELECTED
      AND     M7047  ; NST3_ALL_UNIT_BACK_CLMP_BACK
      ORB
      AND     D5000.0  ; CKT2_AUTO_COTROL
      AND     D7004.7  ; NST3_ANY_FAIL
      AND     L3  ; ALL CONVS RUNNING
      LDI     L1515  ; EMPTYING CYCLE ON OFF
      LD      T641  ; NST3_COMP_PRSNT_EMPTYING_CYCLE
      AND     L1434  ; NST3 COMP PRESENCE SENSOR
      ANI     T638  ; NST3_COMP_NOT_PRSNT_EMPTYING_CYC
      ORB
      ANB
      ANI     L61  ; NST3 BYPASS SEL
      ANI     D7000.4  ; NST3_FAULT_RESET
      ANI     M7049  ; NST3_CYCLE_HOLD
      OUT     D7106.2  ; NST3_AUTO_CYC_READY2
; Rung 77
883   LD      D7009.7  ; NST3_EMERG_RET_COMM
      SET     M7049  ; NST3_CYCLE_HOLD
; Rung 78
891   LDI     D7009.7  ; NST3_EMERG_RET_COMM
      AND     L1402  ; NST3 CYCLE BTN
      RST     M7049  ; NST3_CYCLE_HOLD
; Rung 79
900   LD      L1402  ; NST3 CYCLE BTN
      OUT     T644 K50  ; NST3_STN_CYC_ANTRPT
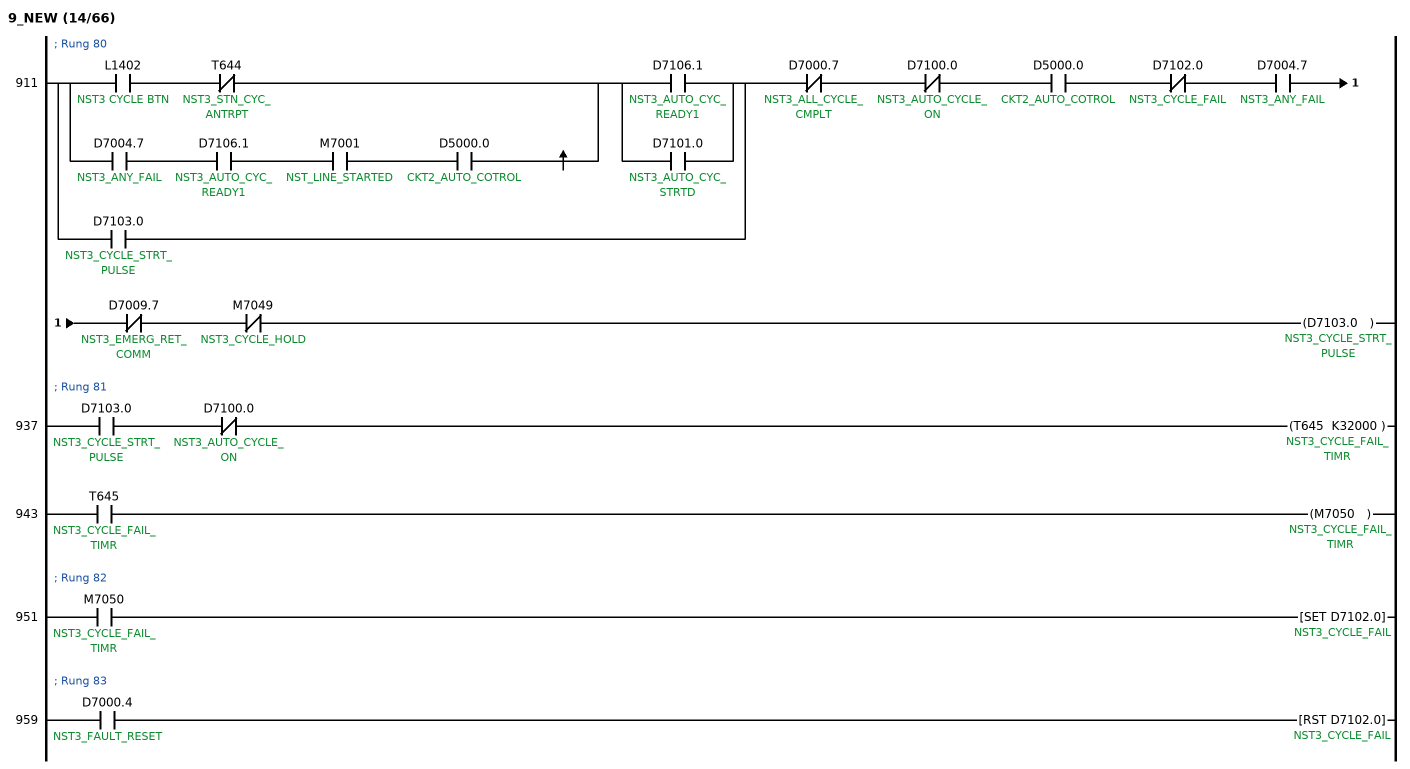
; Rung 80
911   LD      L1402  ; NST3 CYCLE BTN
      ANI     T644  ; NST3_STN_CYC_ANTRPT
      LD      D7004.7  ; NST3_ANY_FAIL
      AND     D7106.1  ; NST3_AUTO_CYC_READY1
      AND     M7001  ; NST_LINE_STARTED
      AND     D5000.0  ; CKT2_AUTO_COTROL
      MEP
      ORB
      LD      D7106.1  ; NST3_AUTO_CYC_READY1
      OR      D7101.0  ; NST3_AUTO_CYC_STRTD
      ANB
      OR      D7103.0  ; NST3_CYCLE_STRT_PULSE
      ANI     D7000.7  ; NST3_ALL_CYCLE_CMPLT
      ANI     D7100.0  ; NST3_AUTO_CYCLE_ON
      AND     D5000.0  ; CKT2_AUTO_COTROL
      ANI     D7102.0  ; NST3_CYCLE_FAIL
      AND     D7004.7  ; NST3_ANY_FAIL
      ANI     D7009.7  ; NST3_EMERG_RET_COMM
      ANI     M7049  ; NST3_CYCLE_HOLD
      OUT     D7103.0  ; NST3_CYCLE_STRT_PULSE
; Rung 81
937   LD      D7103.0  ; NST3_CYCLE_STRT_PULSE
      ANI     D7100.0  ; NST3_AUTO_CYCLE_ON
      OUT     T645 K32000  ; NST3_CYCLE_FAIL_TIMR
943   LD      T645  ; NST3_CYCLE_FAIL_TIMR
      OUT     M7050  ; NST3_CYCLE_FAIL_TIMR
; Rung 82
951   LD      M7050  ; NST3_CYCLE_FAIL_TIMR
      SET     D7102.0  ; NST3_CYCLE_FAIL
; Rung 83
959   LD      D7000.4  ; NST3_FAULT_RESET
      RST     D7102.0  ; NST3_CYCLE_FAIL
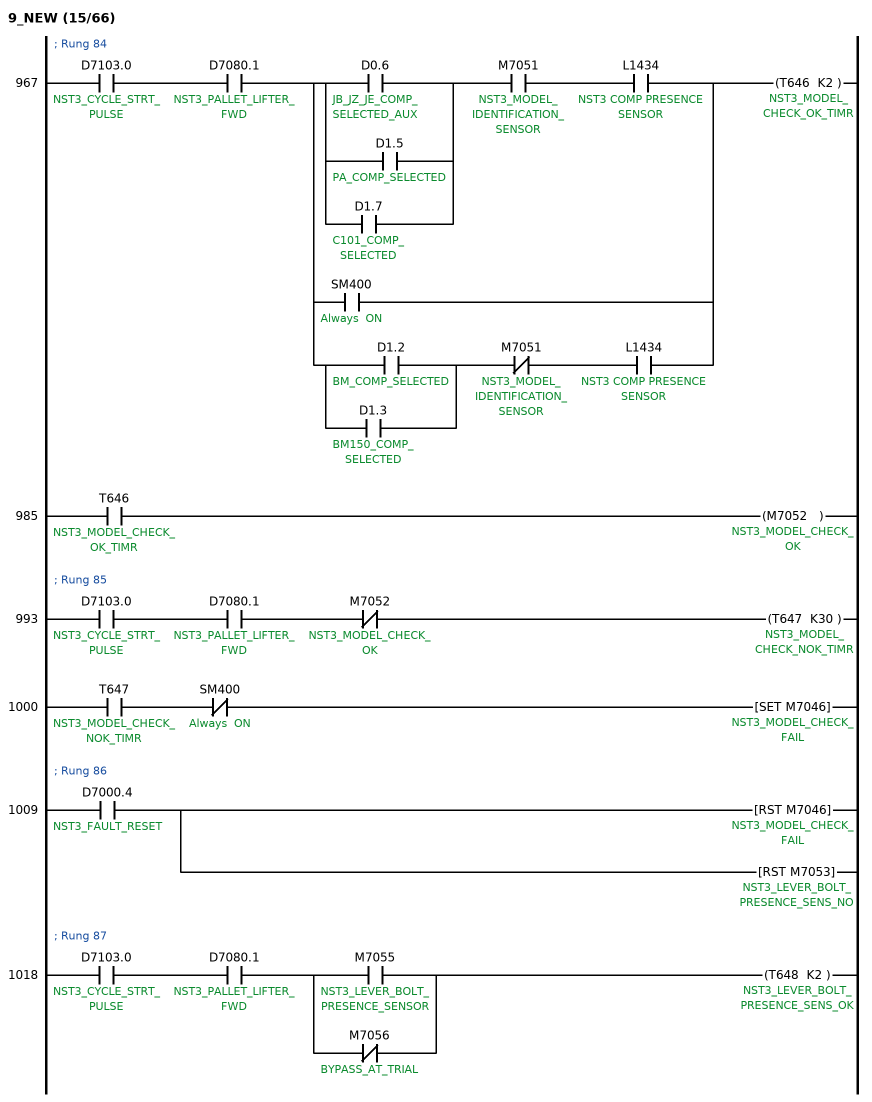
; Rung 84
967   LD      D7103.0  ; NST3_CYCLE_STRT_PULSE
      AND     D7080.1  ; NST3_PALLET_LIFTER_FWD
      LD      D0.6  ; JB_JZ_JE_COMP_SELECTED_AUX
      OR      D1.5  ; PA_COMP_SELECTED
      OR      D1.7  ; C101_COMP_SELECTED
      AND     M7051  ; NST3_MODEL_IDENTIFICATION_SENSOR
      AND     L1434  ; NST3 COMP PRESENCE SENSOR
      OR      SM400  ; Always  ON
      LD      D1.2  ; BM_COMP_SELECTED
      OR      D1.3  ; BM150_COMP_SELECTED
      ANI     M7051  ; NST3_MODEL_IDENTIFICATION_SENSOR
      AND     L1434  ; NST3 COMP PRESENCE SENSOR
      ORB
      ANB
      OUT     T646 K2  ; NST3_MODEL_CHECK_OK_TIMR
985   LD      T646  ; NST3_MODEL_CHECK_OK_TIMR
      OUT     M7052  ; NST3_MODEL_CHECK_OK
; Rung 85
993   LD      D7103.0  ; NST3_CYCLE_STRT_PULSE
      AND     D7080.1  ; NST3_PALLET_LIFTER_FWD
      ANI     M7052  ; NST3_MODEL_CHECK_OK
      OUT     T647 K30  ; NST3_MODEL_CHECK_NOK_TIMR
1000  LD      T647  ; NST3_MODEL_CHECK_NOK_TIMR
      ANI     SM400  ; Always  ON
      SET     M7046  ; NST3_MODEL_CHECK_FAIL
; Rung 86
1009  LD      D7000.4  ; NST3_FAULT_RESET
      RST     M7046  ; NST3_MODEL_CHECK_FAIL
      RST     M7053  ; NST3_LEVER_BOLT_PRESENCE_SENS_NO
; Rung 87
1018  LD      D7103.0  ; NST3_CYCLE_STRT_PULSE
      AND     D7080.1  ; NST3_PALLET_LIFTER_FWD
      LD      M7055  ; NST3_LEVER_BOLT_PRESENCE_SENSOR
      ORI     M7056  ; BYPASS_AT_TRIAL
      ANB
      OUT     T648 K2  ; NST3_LEVER_BOLT_PRESENCE_SENS_OK
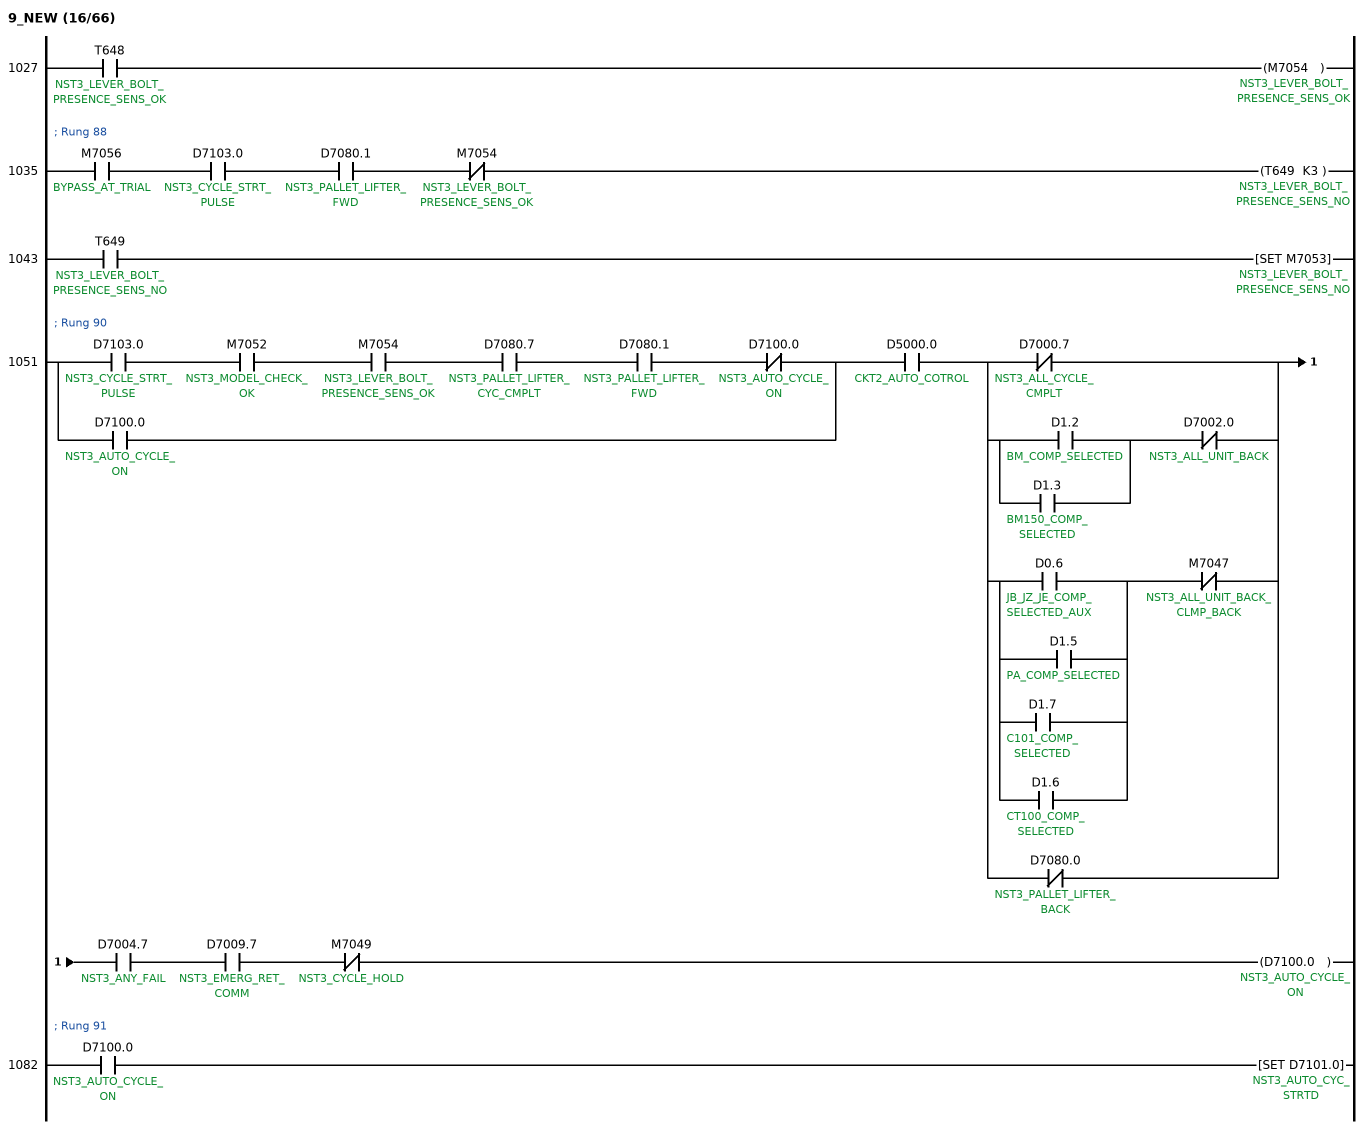
1027  LD      T648  ; NST3_LEVER_BOLT_PRESENCE_SENS_OK
      OUT     M7054  ; NST3_LEVER_BOLT_PRESENCE_SENS_OK
; Rung 88
1035  LD      M7056  ; BYPASS_AT_TRIAL
      AND     D7103.0  ; NST3_CYCLE_STRT_PULSE
      AND     D7080.1  ; NST3_PALLET_LIFTER_FWD
      ANI     M7054  ; NST3_LEVER_BOLT_PRESENCE_SENS_OK
      OUT     T649 K3  ; NST3_LEVER_BOLT_PRESENCE_SENS_NO
1043  LD      T649  ; NST3_LEVER_BOLT_PRESENCE_SENS_NO
      SET     M7053  ; NST3_LEVER_BOLT_PRESENCE_SENS_NO
; Rung 90
1051  LD      D7103.0  ; NST3_CYCLE_STRT_PULSE
      AND     M7052  ; NST3_MODEL_CHECK_OK
      AND     M7054  ; NST3_LEVER_BOLT_PRESENCE_SENS_OK
      AND     D7080.7  ; NST3_PALLET_LIFTER_CYC_CMPLT
      AND     D7080.1  ; NST3_PALLET_LIFTER_FWD
      ANI     D7100.0  ; NST3_AUTO_CYCLE_ON
      OR      D7100.0  ; NST3_AUTO_CYCLE_ON
      AND     D5000.0  ; CKT2_AUTO_COTROL
      LDI     D7000.7  ; NST3_ALL_CYCLE_CMPLT
      LD      D1.2  ; BM_COMP_SELECTED
      OR      D1.3  ; BM150_COMP_SELECTED
      ANI     D7002.0  ; NST3_ALL_UNIT_BACK
      ORB
      LD      D0.6  ; JB_JZ_JE_COMP_SELECTED_AUX
      OR      D1.5  ; PA_COMP_SELECTED
      OR      D1.7  ; C101_COMP_SELECTED
      OR      D1.6  ; CT100_COMP_SELECTED
      ANI     M7047  ; NST3_ALL_UNIT_BACK_CLMP_BACK
      ORB
      ORI     D7080.0  ; NST3_PALLET_LIFTER_BACK
      ANB
      AND     D7004.7  ; NST3_ANY_FAIL
      AND     D7009.7  ; NST3_EMERG_RET_COMM
      ANI     M7049  ; NST3_CYCLE_HOLD
      OUT     D7100.0  ; NST3_AUTO_CYCLE_ON
; Rung 91
1082  LD      D7100.0  ; NST3_AUTO_CYCLE_ON
      SET     D7101.0  ; NST3_AUTO_CYC_STRTD
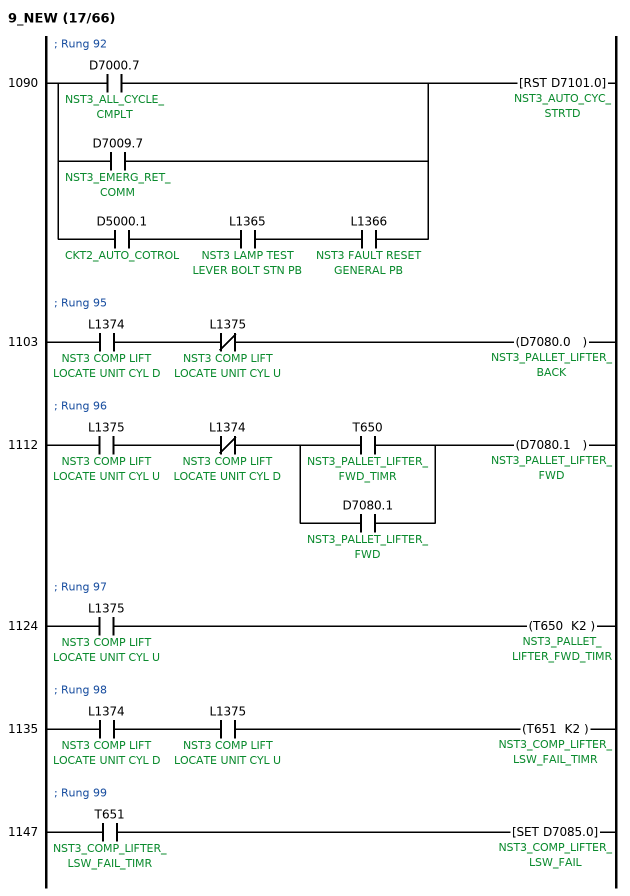
; Rung 92
1090  LD      D7000.7  ; NST3_ALL_CYCLE_CMPLT
      OR      D7009.7  ; NST3_EMERG_RET_COMM
      LD      D5000.1  ; CKT2_AUTO_COTROL
      AND     L1365  ; NST3 LAMP TEST LEVER BOLT STN PB
      AND     L1366  ; NST3 FAULT RESET GENERAL PB
      ORB
      RST     D7101.0  ; NST3_AUTO_CYC_STRTD
; Rung 95
1103  LD      L1374  ; NST3 COMP LIFT LOCATE UNIT CYL D
      ANI     L1375  ; NST3 COMP LIFT LOCATE UNIT CYL U
      OUT     D7080.0  ; NST3_PALLET_LIFTER_BACK
; Rung 96
1112  LD      L1375  ; NST3 COMP LIFT LOCATE UNIT CYL U
      ANI     L1374  ; NST3 COMP LIFT LOCATE UNIT CYL D
      LD      T650  ; NST3_PALLET_LIFTER_FWD_TIMR
      OR      D7080.1  ; NST3_PALLET_LIFTER_FWD
      ANB
      OUT     D7080.1  ; NST3_PALLET_LIFTER_FWD
; Rung 97
1124  LD      L1375  ; NST3 COMP LIFT LOCATE UNIT CYL U
      OUT     T650 K2  ; NST3_PALLET_LIFTER_FWD_TIMR
; Rung 98
1135  LD      L1374  ; NST3 COMP LIFT LOCATE UNIT CYL D
      AND     L1375  ; NST3 COMP LIFT LOCATE UNIT CYL U
      OUT     T651 K2  ; NST3_COMP_LIFTER_LSW_FAIL_TIMR
; Rung 99
1147  LD      T651  ; NST3_COMP_LIFTER_LSW_FAIL_TIMR
      SET     D7085.0  ; NST3_COMP_LIFTER_LSW_FAIL
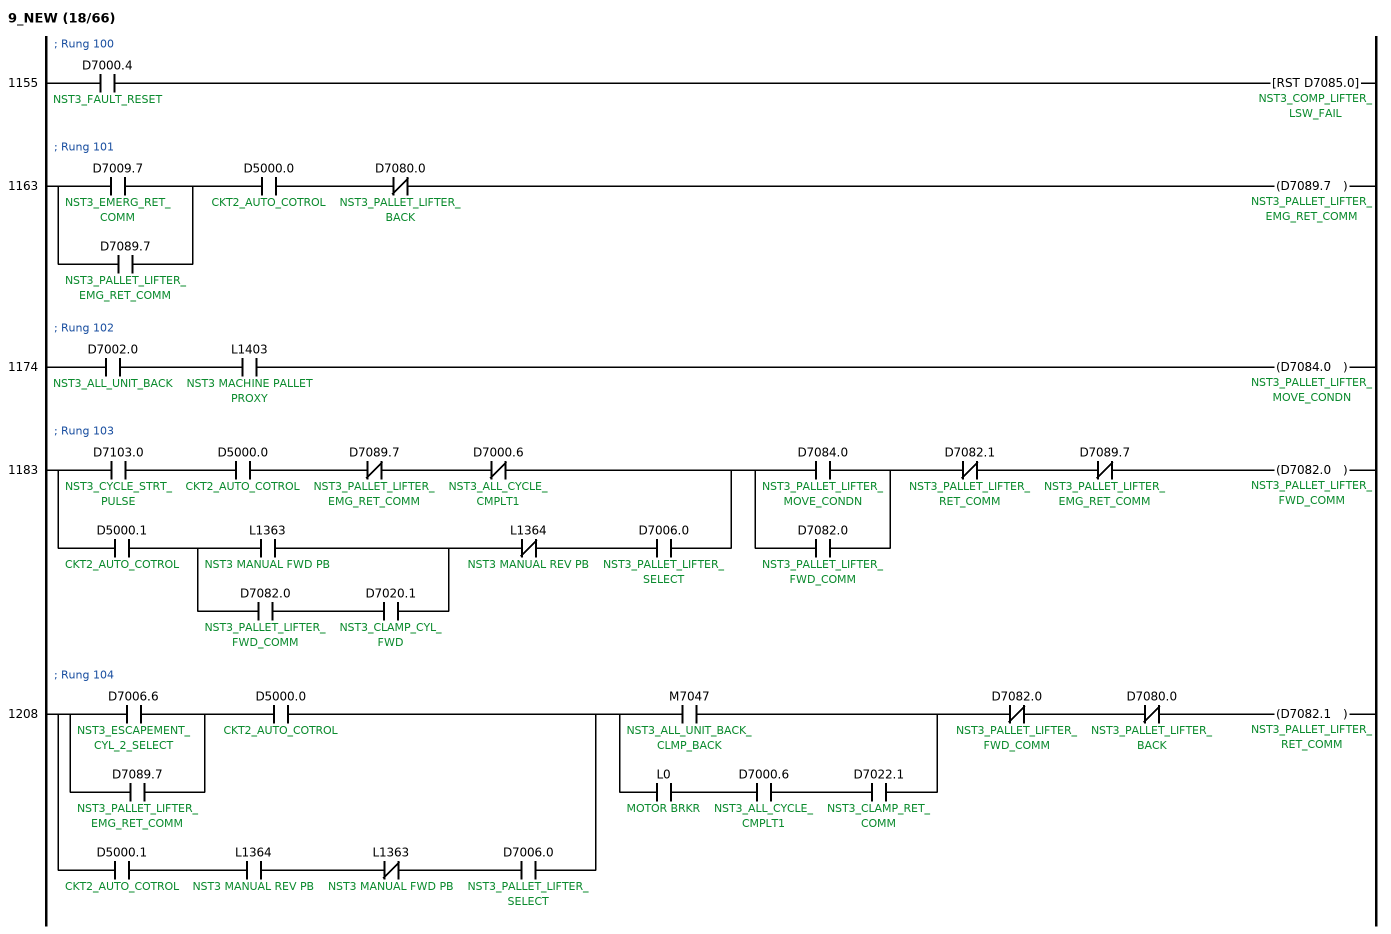
; Rung 100
1155  LD      D7000.4  ; NST3_FAULT_RESET
      RST     D7085.0  ; NST3_COMP_LIFTER_LSW_FAIL
; Rung 101
1163  LD      D7009.7  ; NST3_EMERG_RET_COMM
      OR      D7089.7  ; NST3_PALLET_LIFTER_EMG_RET_COMM
      AND     D5000.0  ; CKT2_AUTO_COTROL
      ANI     D7080.0  ; NST3_PALLET_LIFTER_BACK
      OUT     D7089.7  ; NST3_PALLET_LIFTER_EMG_RET_COMM
; Rung 102
1174  LD      D7002.0  ; NST3_ALL_UNIT_BACK
      AND     L1403  ; NST3 MACHINE PALLET PROXY
      OUT     D7084.0  ; NST3_PALLET_LIFTER_MOVE_CONDN
; Rung 103
1183  LD      D7103.0  ; NST3_CYCLE_STRT_PULSE
      AND     D5000.0  ; CKT2_AUTO_COTROL
      ANI     D7089.7  ; NST3_PALLET_LIFTER_EMG_RET_COMM
      ANI     D7000.6  ; NST3_ALL_CYCLE_CMPLT1
      LD      D5000.1  ; CKT2_AUTO_COTROL
      LD      L1363  ; NST3 MANUAL FWD PB
      LD      D7082.0  ; NST3_PALLET_LIFTER_FWD_COMM
      AND     D7020.1  ; NST3_CLAMP_CYL_FWD
      ORB
      ANB
      ANI     L1364  ; NST3 MANUAL REV PB
      AND     D7006.0  ; NST3_PALLET_LIFTER_SELECT
      ORB
      LD      D7084.0  ; NST3_PALLET_LIFTER_MOVE_CONDN
      OR      D7082.0  ; NST3_PALLET_LIFTER_FWD_COMM
      ANB
      ANI     D7082.1  ; NST3_PALLET_LIFTER_RET_COMM
      ANI     D7089.7  ; NST3_PALLET_LIFTER_EMG_RET_COMM
      OUT     D7082.0  ; NST3_PALLET_LIFTER_FWD_COMM
; Rung 104
1208  LD      D7006.6  ; NST3_ESCAPEMENT_CYL_2_SELECT
      OR      D7089.7  ; NST3_PALLET_LIFTER_EMG_RET_COMM
      AND     D5000.0  ; CKT2_AUTO_COTROL
      LD      D5000.1  ; CKT2_AUTO_COTROL
      AND     L1364  ; NST3 MANUAL REV PB
      ANI     L1363  ; NST3 MANUAL FWD PB
      AND     D7006.0  ; NST3_PALLET_LIFTER_SELECT
      ORB
      LD      M7047  ; NST3_ALL_UNIT_BACK_CLMP_BACK
      LD      L0  ; MOTOR BRKR
      AND     D7000.6  ; NST3_ALL_CYCLE_CMPLT1
      AND     D7022.1  ; NST3_CLAMP_RET_COMM
      ORB
      ANB
      ANI     D7082.0  ; NST3_PALLET_LIFTER_FWD_COMM
      ANI     D7080.0  ; NST3_PALLET_LIFTER_BACK
      OUT     D7082.1  ; NST3_PALLET_LIFTER_RET_COMM
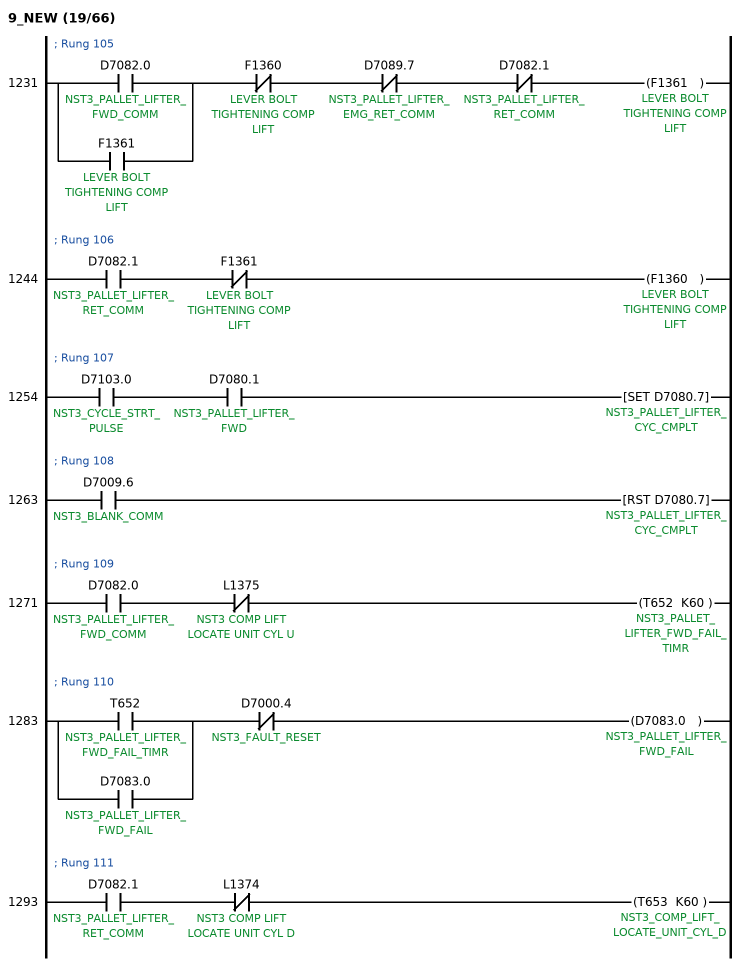
; Rung 105
1231  LD      D7082.0  ; NST3_PALLET_LIFTER_FWD_COMM
      OR      F1361  ; LEVER BOLT TIGHTENING COMP LIFT
      ANI     F1360  ; LEVER BOLT TIGHTENING COMP LIFT
      ANI     D7089.7  ; NST3_PALLET_LIFTER_EMG_RET_COMM
      ANI     D7082.1  ; NST3_PALLET_LIFTER_RET_COMM
      OUT     F1361  ; LEVER BOLT TIGHTENING COMP LIFT
; Rung 106
1244  LD      D7082.1  ; NST3_PALLET_LIFTER_RET_COMM
      ANI     F1361  ; LEVER BOLT TIGHTENING COMP LIFT
      OUT     F1360  ; LEVER BOLT TIGHTENING COMP LIFT
; Rung 107
1254  LD      D7103.0  ; NST3_CYCLE_STRT_PULSE
      AND     D7080.1  ; NST3_PALLET_LIFTER_FWD
      SET     D7080.7  ; NST3_PALLET_LIFTER_CYC_CMPLT
; Rung 108
1263  LD      D7009.6  ; NST3_BLANK_COMM
      RST     D7080.7  ; NST3_PALLET_LIFTER_CYC_CMPLT
; Rung 109
1271  LD      D7082.0  ; NST3_PALLET_LIFTER_FWD_COMM
      ANI     L1375  ; NST3 COMP LIFT LOCATE UNIT CYL U
      OUT     T652 K60  ; NST3_PALLET_LIFTER_FWD_FAIL_TIMR
; Rung 110
1283  LD      T652  ; NST3_PALLET_LIFTER_FWD_FAIL_TIMR
      OR      D7083.0  ; NST3_PALLET_LIFTER_FWD_FAIL
      ANI     D7000.4  ; NST3_FAULT_RESET
      OUT     D7083.0  ; NST3_PALLET_LIFTER_FWD_FAIL
; Rung 111
1293  LD      D7082.1  ; NST3_PALLET_LIFTER_RET_COMM
      ANI     L1374  ; NST3 COMP LIFT LOCATE UNIT CYL D
      OUT     T653 K60  ; NST3_COMP_LIFT_LOCATE_UNIT_CYL_D
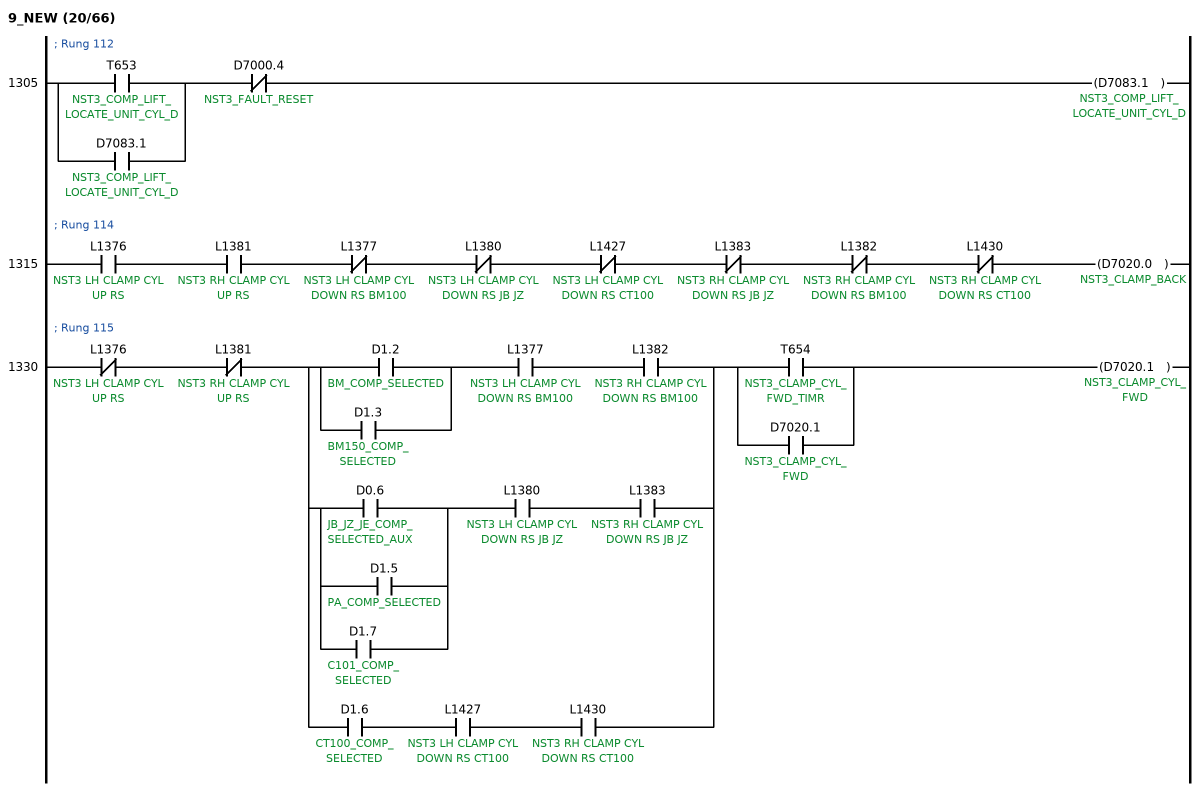
; Rung 112
1305  LD      T653  ; NST3_COMP_LIFT_LOCATE_UNIT_CYL_D
      OR      D7083.1  ; NST3_COMP_LIFT_LOCATE_UNIT_CYL_D
      ANI     D7000.4  ; NST3_FAULT_RESET
      OUT     D7083.1  ; NST3_COMP_LIFT_LOCATE_UNIT_CYL_D
; Rung 114
1315  LD      L1376  ; NST3 LH CLAMP CYL UP RS
      AND     L1381  ; NST3 RH CLAMP CYL UP RS
      ANI     L1377  ; NST3 LH CLAMP CYL DOWN RS BM100
      ANI     L1380  ; NST3 LH CLAMP CYL DOWN RS JB JZ
      ANI     L1427  ; NST3 LH CLAMP CYL DOWN RS CT100
      ANI     L1383  ; NST3 RH CLAMP CYL DOWN RS JB JZ
      ANI     L1382  ; NST3 RH CLAMP CYL DOWN RS BM100
      ANI     L1430  ; NST3 RH CLAMP CYL DOWN RS CT100
      OUT     D7020.0  ; NST3_CLAMP_BACK
; Rung 115
1330  LDI     L1376  ; NST3 LH CLAMP CYL UP RS
      ANI     L1381  ; NST3 RH CLAMP CYL UP RS
      LD      D1.2  ; BM_COMP_SELECTED
      OR      D1.3  ; BM150_COMP_SELECTED
      AND     L1377  ; NST3 LH CLAMP CYL DOWN RS BM100
      AND     L1382  ; NST3 RH CLAMP CYL DOWN RS BM100
      LD      D0.6  ; JB_JZ_JE_COMP_SELECTED_AUX
      OR      D1.5  ; PA_COMP_SELECTED
      OR      D1.7  ; C101_COMP_SELECTED
      AND     L1380  ; NST3 LH CLAMP CYL DOWN RS JB JZ
      AND     L1383  ; NST3 RH CLAMP CYL DOWN RS JB JZ
      ORB
      LD      D1.6  ; CT100_COMP_SELECTED
      AND     L1427  ; NST3 LH CLAMP CYL DOWN RS CT100
      AND     L1430  ; NST3 RH CLAMP CYL DOWN RS CT100
      ORB
      ANB
      LD      T654  ; NST3_CLAMP_CYL_FWD_TIMR
      OR      D7020.1  ; NST3_CLAMP_CYL_FWD
      ANB
      OUT     D7020.1  ; NST3_CLAMP_CYL_FWD
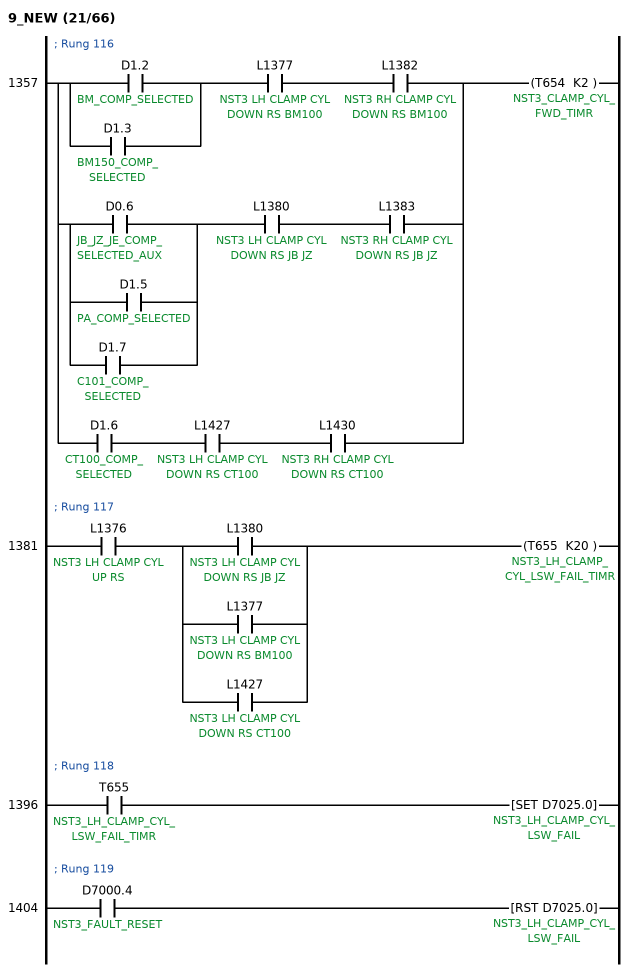
; Rung 116
1357  LD      D1.2  ; BM_COMP_SELECTED
      OR      D1.3  ; BM150_COMP_SELECTED
      AND     L1377  ; NST3 LH CLAMP CYL DOWN RS BM100
      AND     L1382  ; NST3 RH CLAMP CYL DOWN RS BM100
      LD      D0.6  ; JB_JZ_JE_COMP_SELECTED_AUX
      OR      D1.5  ; PA_COMP_SELECTED
      OR      D1.7  ; C101_COMP_SELECTED
      AND     L1380  ; NST3 LH CLAMP CYL DOWN RS JB JZ
      AND     L1383  ; NST3 RH CLAMP CYL DOWN RS JB JZ
      ORB
      LD      D1.6  ; CT100_COMP_SELECTED
      AND     L1427  ; NST3 LH CLAMP CYL DOWN RS CT100
      AND     L1430  ; NST3 RH CLAMP CYL DOWN RS CT100
      ORB
      OUT     T654 K2  ; NST3_CLAMP_CYL_FWD_TIMR
; Rung 117
1381  LD      L1376  ; NST3 LH CLAMP CYL UP RS
      LD      L1380  ; NST3 LH CLAMP CYL DOWN RS JB JZ
      OR      L1377  ; NST3 LH CLAMP CYL DOWN RS BM100
      OR      L1427  ; NST3 LH CLAMP CYL DOWN RS CT100
      ANB
      OUT     T655 K20  ; NST3_LH_CLAMP_CYL_LSW_FAIL_TIMR
; Rung 118
1396  LD      T655  ; NST3_LH_CLAMP_CYL_LSW_FAIL_TIMR
      SET     D7025.0  ; NST3_LH_CLAMP_CYL_LSW_FAIL
; Rung 119
1404  LD      D7000.4  ; NST3_FAULT_RESET
      RST     D7025.0  ; NST3_LH_CLAMP_CYL_LSW_FAIL
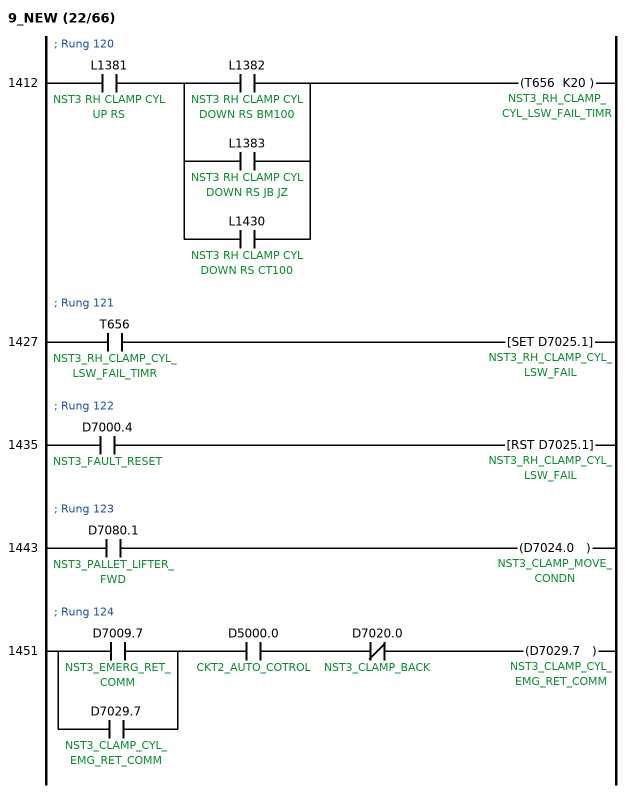
; Rung 120
1412  LD      L1381  ; NST3 RH CLAMP CYL UP RS
      LD      L1382  ; NST3 RH CLAMP CYL DOWN RS BM100
      OR      L1383  ; NST3 RH CLAMP CYL DOWN RS JB JZ
      OR      L1430  ; NST3 RH CLAMP CYL DOWN RS CT100
      ANB
      OUT     T656 K20  ; NST3_RH_CLAMP_CYL_LSW_FAIL_TIMR
; Rung 121
1427  LD      T656  ; NST3_RH_CLAMP_CYL_LSW_FAIL_TIMR
      SET     D7025.1  ; NST3_RH_CLAMP_CYL_LSW_FAIL
; Rung 122
1435  LD      D7000.4  ; NST3_FAULT_RESET
      RST     D7025.1  ; NST3_RH_CLAMP_CYL_LSW_FAIL
; Rung 123
1443  LD      D7080.1  ; NST3_PALLET_LIFTER_FWD
      OUT     D7024.0  ; NST3_CLAMP_MOVE_CONDN
; Rung 124
1451  LD      D7009.7  ; NST3_EMERG_RET_COMM
      OR      D7029.7  ; NST3_CLAMP_CYL_EMG_RET_COMM
      AND     D5000.0  ; CKT2_AUTO_COTROL
      ANI     D7020.0  ; NST3_CLAMP_BACK
      OUT     D7029.7  ; NST3_CLAMP_CYL_EMG_RET_COMM
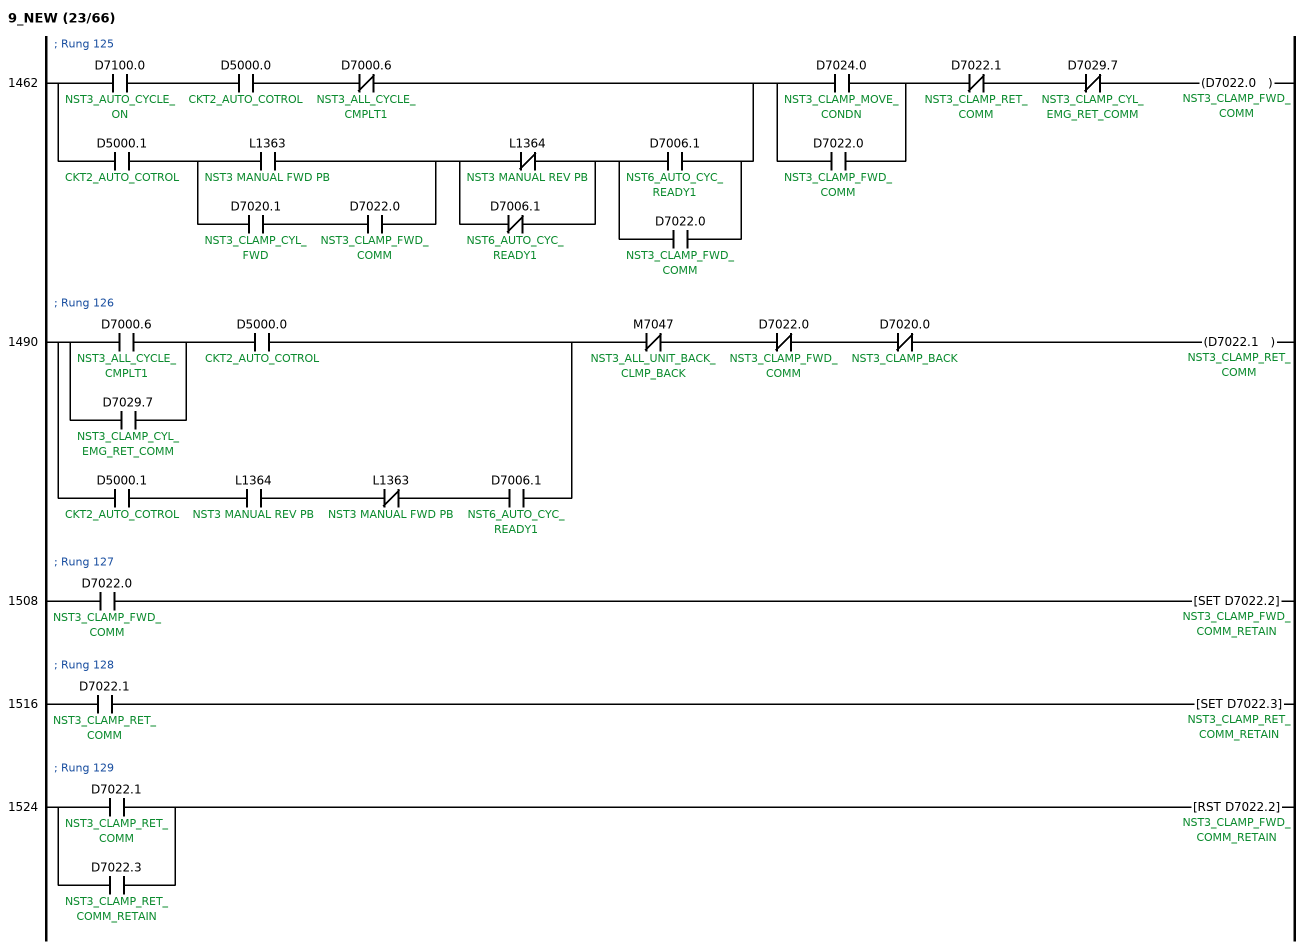
; Rung 125
1462  LD      D7100.0  ; NST3_AUTO_CYCLE_ON
      AND     D5000.0  ; CKT2_AUTO_COTROL
      ANI     D7000.6  ; NST3_ALL_CYCLE_CMPLT1
      LD      D5000.1  ; CKT2_AUTO_COTROL
      LD      L1363  ; NST3 MANUAL FWD PB
      LD      D7020.1  ; NST3_CLAMP_CYL_FWD
      AND     D7022.0  ; NST3_CLAMP_FWD_COMM
      ORB
      ANB
      LDI     L1364  ; NST3 MANUAL REV PB
      ORI     D7006.1  ; NST6_AUTO_CYC_READY1
      ANB
      LD      D7006.1  ; NST6_AUTO_CYC_READY1
      OR      D7022.0  ; NST3_CLAMP_FWD_COMM
      ANB
      ORB
      LD      D7024.0  ; NST3_CLAMP_MOVE_CONDN
      OR      D7022.0  ; NST3_CLAMP_FWD_COMM
      ANB
      ANI     D7022.1  ; NST3_CLAMP_RET_COMM
      ANI     D7029.7  ; NST3_CLAMP_CYL_EMG_RET_COMM
      OUT     D7022.0  ; NST3_CLAMP_FWD_COMM
; Rung 126
1490  LD      D7000.6  ; NST3_ALL_CYCLE_CMPLT1
      OR      D7029.7  ; NST3_CLAMP_CYL_EMG_RET_COMM
      AND     D5000.0  ; CKT2_AUTO_COTROL
      LD      D5000.1  ; CKT2_AUTO_COTROL
      AND     L1364  ; NST3 MANUAL REV PB
      ANI     L1363  ; NST3 MANUAL FWD PB
      AND     D7006.1  ; NST6_AUTO_CYC_READY1
      ORB
      ANI     M7047  ; NST3_ALL_UNIT_BACK_CLMP_BACK
      ANI     D7022.0  ; NST3_CLAMP_FWD_COMM
      ANI     D7020.0  ; NST3_CLAMP_BACK
      OUT     D7022.1  ; NST3_CLAMP_RET_COMM
; Rung 127
1508  LD      D7022.0  ; NST3_CLAMP_FWD_COMM
      SET     D7022.2  ; NST3_CLAMP_FWD_COMM_RETAIN
; Rung 128
1516  LD      D7022.1  ; NST3_CLAMP_RET_COMM
      SET     D7022.3  ; NST3_CLAMP_RET_COMM_RETAIN
; Rung 129
1524  LD      D7022.1  ; NST3_CLAMP_RET_COMM
      OR      D7022.3  ; NST3_CLAMP_RET_COMM_RETAIN
      RST     D7022.2  ; NST3_CLAMP_FWD_COMM_RETAIN
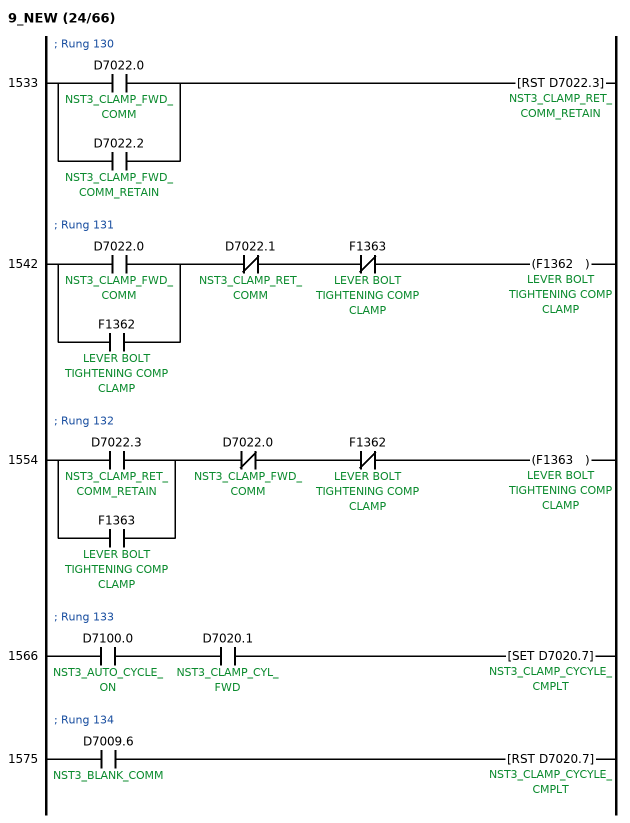
; Rung 130
1533  LD      D7022.0  ; NST3_CLAMP_FWD_COMM
      OR      D7022.2  ; NST3_CLAMP_FWD_COMM_RETAIN
      RST     D7022.3  ; NST3_CLAMP_RET_COMM_RETAIN
; Rung 131
1542  LD      D7022.0  ; NST3_CLAMP_FWD_COMM
      OR      F1362  ; LEVER BOLT TIGHTENING COMP CLAMP
      ANI     D7022.1  ; NST3_CLAMP_RET_COMM
      ANI     F1363  ; LEVER BOLT TIGHTENING COMP CLAMP
      OUT     F1362  ; LEVER BOLT TIGHTENING COMP CLAMP
; Rung 132
1554  LD      D7022.3  ; NST3_CLAMP_RET_COMM_RETAIN
      OR      F1363  ; LEVER BOLT TIGHTENING COMP CLAMP
      ANI     D7022.0  ; NST3_CLAMP_FWD_COMM
      ANI     F1362  ; LEVER BOLT TIGHTENING COMP CLAMP
      OUT     F1363  ; LEVER BOLT TIGHTENING COMP CLAMP
; Rung 133
1566  LD      D7100.0  ; NST3_AUTO_CYCLE_ON
      AND     D7020.1  ; NST3_CLAMP_CYL_FWD
      SET     D7020.7  ; NST3_CLAMP_CYCYLE_CMPLT
; Rung 134
1575  LD      D7009.6  ; NST3_BLANK_COMM
      RST     D7020.7  ; NST3_CLAMP_CYCYLE_CMPLT
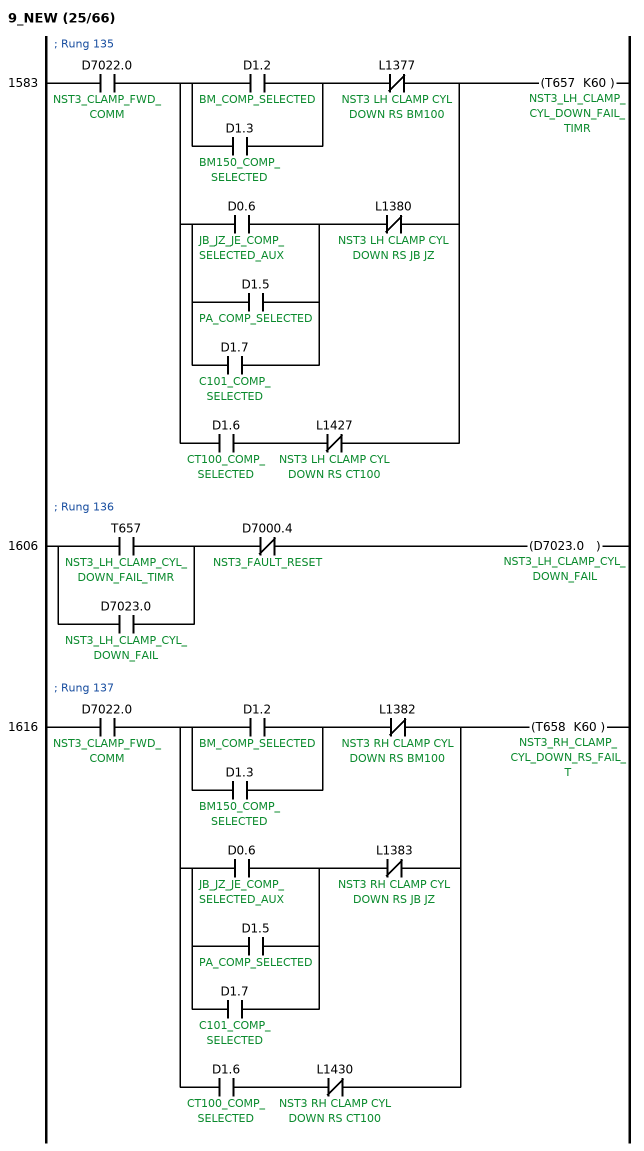
; Rung 135
1583  LD      D7022.0  ; NST3_CLAMP_FWD_COMM
      LD      D1.2  ; BM_COMP_SELECTED
      OR      D1.3  ; BM150_COMP_SELECTED
      ANI     L1377  ; NST3 LH CLAMP CYL DOWN RS BM100
      LD      D0.6  ; JB_JZ_JE_COMP_SELECTED_AUX
      OR      D1.5  ; PA_COMP_SELECTED
      OR      D1.7  ; C101_COMP_SELECTED
      ANI     L1380  ; NST3 LH CLAMP CYL DOWN RS JB JZ
      ORB
      LD      D1.6  ; CT100_COMP_SELECTED
      ANI     L1427  ; NST3 LH CLAMP CYL DOWN RS CT100
      ORB
      ANB
      OUT     T657 K60  ; NST3_LH_CLAMP_CYL_DOWN_FAIL_TIMR
; Rung 136
1606  LD      T657  ; NST3_LH_CLAMP_CYL_DOWN_FAIL_TIMR
      OR      D7023.0  ; NST3_LH_CLAMP_CYL_DOWN_FAIL
      ANI     D7000.4  ; NST3_FAULT_RESET
      OUT     D7023.0  ; NST3_LH_CLAMP_CYL_DOWN_FAIL
; Rung 137
1616  LD      D7022.0  ; NST3_CLAMP_FWD_COMM
      LD      D1.2  ; BM_COMP_SELECTED
      OR      D1.3  ; BM150_COMP_SELECTED
      ANI     L1382  ; NST3 RH CLAMP CYL DOWN RS BM100
      LD      D0.6  ; JB_JZ_JE_COMP_SELECTED_AUX
      OR      D1.5  ; PA_COMP_SELECTED
      OR      D1.7  ; C101_COMP_SELECTED
      ANI     L1383  ; NST3 RH CLAMP CYL DOWN RS JB JZ
      ORB
      LD      D1.6  ; CT100_COMP_SELECTED
      ANI     L1430  ; NST3 RH CLAMP CYL DOWN RS CT100
      ORB
      ANB
      OUT     T658 K60  ; NST3_RH_CLAMP_CYL_DOWN_RS_FAIL_T
